LIN {X 0,Y 575.893,Z 1106.128,A -85,B 0,C 180,E1 20228.402,E2 20228.402} C_VEL
LIN {X 0,Y 578.191,Z 1090.768,A -85,B 0,C 180,E1 20226.346,E2 20226.346} C_VEL
LIN {X 0,Y 580.577,Z 1075.313,A -85,B 0,C 180,E1 20224.483,E2 20224.483} C_VEL
LIN {X 0,Y 583.778,Z 1055.461,A -85,B 0,C 180,E1 20222.344,E2 20222.344} C_VEL
LIN {X 0,Y 586.979,Z 1035.406,A -85,B 0,C 180,E1 20220.459,E2 20220.459} C_VEL
LIN {X 0,Y 589.808,Z 1017.804,A -85,B 0,C 180,E1 20218.978,E2 20218.978} C_VEL
LIN {X 0,Y 592.773,Z 999.025,A -85,B 0,C 180,E1 20217.561,E2 20217.561} C_VEL
LIN {X 0,Y 596.383,Z 975.656,A -85,B 0,C 180,E1 20216.004,E2 20216.004} C_VEL
LIN {X 0,Y 599.713,Z 951.946,A -85,B 0,C 180,E1 20214.652,E2 20214.652} C_VEL
LIN {X 0,Y 602.211,Z 933.032,A -85,B 0,C 180,E1 20213.707,E2 20213.707} C_VEL
LIN {X 0,Y 604.654,Z 912.644,A -85,B 0,C 180,E1 20212.814,E2 20212.814} C_VEL
LIN {X 0,Y 607.042,Z 890.934,A -85,B 0,C 180,E1 20212.003,E2 20212.003} C_VEL
LIN {X 0,Y 609.575,Z 864.282,A -85,B 0,C 180,E1 20211.183,E2 20211.183} C_VEL
LIN {X 0,Y 611.456,Z 838.408,A -85,B 0,C 180,E1 20210.573,E2 20210.573} C_VEL
LIN {X 0,Y 612.734,Z 815.587,A -85,B 0,C 180,E1 20210.167,E2 20210.167} C_VEL
LIN {X 0,Y 618.857,Z 603.625,A -85,B 0,C 180,E1 20207.181,E2 20207.181} C_VEL
LIN {X 0,Y 624.347,Z 417.468,A -85,B 0,C 180,E1 20204.512,E2 20204.512} C_VEL
LIN {X 0,Y 610.025,Z 396.851,A -85,B 0,C 180,E1 20202.474,E2 20202.474} C_VEL
LIN {X 0,Y 593.081,Z 373.946,A -85,B 0,C 180,E1 20199.872,E2 20199.872} C_VEL
LIN {X 0,Y 586.63,Z 365.779,A -85,B 0,C 180,E1 20198.816,E2 20198.816} C_VEL
LIN {X 0,Y 582.842,Z 360.939,A -85,B 0,C 180,E1 20198.172,E2 20198.172} C_VEL
LIN {X 0,Y 579.584,Z 357.07,A -85,B 0,C 180,E1 20197.61,E2 20197.61} C_VEL
LIN {X 0,Y 578.5,Z 355.414,A -85,B 0,C 180,E1 20197.412,E2 20197.412} C_VEL
LIN {X 0,Y 575.382,Z 352.205,A -85,B 0,C 180,E1 20196.868,E2 20196.868} C_VEL
LIN {X 0,Y 573.879,Z 349.556,A -85,B 0,C 180,E1 20196.576,E2 20196.576} C_VEL
LIN {X 0,Y 571.012,Z 347.283,A -85,B 0,C 180,E1 20196.072,E2 20196.072} C_VEL
LIN {X 0,Y 569.539,Z 344.267,A -85,B 0,C 180,E1 20195.766,E2 20195.766} C_VEL
LIN {X 0,Y 569.361,Z 343.303,A -85,B 0,C 180,E1 20195.707,E2 20195.707} C_VEL
LIN {X 0,Y 569.351,Z 343.308,A -85,B 0,C 180,E1 20192.358,E2 20192.358} C_VEL
LIN {X 0,Y 569.387,Z 343.308,A -85,B 0,C 180,E1 20189.107,E2 20189.107} C_VEL
LIN {X 0,Y 569.334,Z 343.259,A -85,B 0,C 180,E1 20185.82,E2 20185.82} C_VEL
LIN {X 0,Y 569.37,Z 343.294,A -85,B 0,C 180,E1 20182.51,E2 20182.51} C_VEL
LIN {X 0,Y 569.339,Z 343.26,A -85,B 0,C 180,E1 20179.386,E2 20179.386} C_VEL
LIN {X 0,Y 569.332,Z 343.299,A -85,B 0,C 180,E1 20176.006,E2 20176.006} C_VEL
LIN {X 0,Y 569.365,Z 343.249,A -85,B 0,C 180,E1 20172.887,E2 20172.887} C_VEL
LIN {X 0,Y 569.32,Z 343.309,A -85,B 0,C 180,E1 20169.707,E2 20169.707} C_VEL
LIN {X 0,Y 569.387,Z 343.308,A -85,B 0,C 180,E1 20166.554,E2 20166.554} C_VEL
LIN {X 0,Y 569.312,Z 343.314,A -85,B 0,C 180,E1 20163.323,E2 20163.323} C_VEL
LIN {X 0,Y 569.356,Z 343.31,A -85,B 0,C 180,E1 20160.101,E2 20160.101} C_VEL
LIN {X 0,Y 569.307,Z 343.31,A -85,B 0,C 180,E1 20157.08,E2 20157.08} C_VEL
LIN {X 0,Y 569.321,Z 343.308,A -85,B 0,C 180,E1 20153.745,E2 20153.745} C_VEL
LIN {X 0,Y 569.3,Z 343.302,A -85,B 0,C 180,E1 20150.905,E2 20150.905} C_VEL
LIN {X 0,Y 569.305,Z 343.271,A -85,B 0,C 180,E1 20147.557,E2 20147.557} C_VEL
LIN {X 0,Y 569.299,Z 343.289,A -85,B 0,C 180,E1 20144.628,E2 20144.628} C_VEL
LIN {X 0,Y 569.287,Z 343.271,A -85,B 0,C 180,E1 20141.251,E2 20141.251} C_VEL
LIN {X 0,Y 569.315,Z 343.302,A -85,B 0,C 180,E1 20138.248,E2 20138.248} C_VEL
LIN {X 0,Y 569.275,Z 343.263,A -85,B 0,C 180,E1 20135,E2 20135} C_VEL
LIN {X 0,Y 569.359,Z 343.305,A -85,B 0,C 180,E1 20131.809,E2 20131.809} C_VEL
LIN {X 0,Y 569.297,Z 343.395,A -85,B 0,C 180,E1 20130.946,E2 20130.946} C_VEL
LIN {X 0,Y 570.439,Z 346.544,A -85,B 0,C 180,E1 20130.376,E2 20130.376} C_VEL
LIN {X 0,Y 571.962,Z 348.62,A -85,B 0,C 180,E1 20129.886,E2 20129.886} C_VEL
LIN {X 0,Y 574.856,Z 352.888,A -85,B 0,C 180,E1 20129.302,E2 20129.302} C_VEL
LIN {X 0,Y 577.63,Z 356.406,A -85,B 0,C 180,E1 20128.801,E2 20128.801} C_VEL
LIN {X 0,Y 584.527,Z 365.235,A -85,B 0,C 180,E1 20127.599,E2 20127.599} C_VEL
LIN {X 0,Y 592.875,Z 376.369,A -85,B 0,C 180,E1 20126.211,E2 20126.211} C_VEL
LIN {X 0,Y 606.926,Z 395.613,A -85,B 0,C 180,E1 20124.033,E2 20124.033} C_VEL
LIN {X 0,Y 619.297,Z 413.266,A -85,B 0,C 180,E1 20122.242,E2 20122.242} C_VEL
LIN {X 0,Y 624.456,Z 421.081,A -85,B 0,C 180,E1 20121.519,E2 20121.519} C_VEL
LIN {X 0,Y 618.456,Z 624.273,A -85,B 0,C 180,E1 20118.616,E2 20118.616} C_VEL
LIN {X 0,Y 612.63,Z 826.368,A -85,B 0,C 180,E1 20115.769,E2 20115.769} C_VEL
LIN {X 0,Y 611.284,Z 850.031,A -85,B 0,C 180,E1 20115.341,E2 20115.341} C_VEL
LIN {X 0,Y 609.041,Z 878.855,A -85,B 0,C 180,E1 20114.633,E2 20114.633} C_VEL
LIN {X 0,Y 606.975,Z 900.549,A -85,B 0,C 180,E1 20113.955,E2 20113.955} C_VEL
LIN {X 0,Y 604.717,Z 921.391,A -85,B 0,C 180,E1 20113.181,E2 20113.181} C_VEL
LIN {X 0,Y 602.477,Z 940.397,A -85,B 0,C 180,E1 20112.361,E2 20112.361} C_VEL
LIN {X 0,Y 599.946,Z 959.808,A -85,B 0,C 180,E1 20111.411,E2 20111.411} C_VEL
LIN {X 0,Y 597.021,Z 980.896,A -85,B 0,C 180,E1 20110.234,E2 20110.234} C_VEL
LIN {X 0,Y 593.329,Z 1005.625,A -85,B 0,C 180,E1 20108.636,E2 20108.636} C_VEL
LIN {X 0,Y 590.183,Z 1025.543,A -85,B 0,C 180,E1 20107.155,E2 20107.155} C_VEL
LIN {X 0,Y 587.381,Z 1042.971,A -85,B 0,C 180,E1 20105.709,E2 20105.709} C_VEL
LIN {X 0,Y 584.603,Z 1060.16,A -85,B 0,C 180,E1 20104.124,E2 20104.124} C_VEL
LIN {X 0,Y 581.464,Z 1079.866,A -85,B 0,C 180,E1 20102.097,E2 20102.097} C_VEL
LIN {X 0,Y 578.617,Z 1097.979,A -85,B 0,C 180,E1 20099.961,E2 20099.961} C_VEL
LIN {X 0,Y 576.364,Z 1112.967,A -85,B 0,C 180,E1 20097.99,E2 20097.99} C_VEL
LIN {X 0,Y 574.255,Z 1127.876,A -85,B 0,C 180,E1 20095.804,E2 20095.804} C_VEL
LIN {X 0,Y 572.237,Z 1143.699,A -85,B 0,C 180,E1 20093.151,E2 20093.151} C_VEL
LIN {X 0,Y 570.921,Z 1155.261,A -85,B 0,C 180,E1 20090.933,E2 20090.933} C_VEL
LIN {X 0,Y 569.926,Z 1165.441,A -85,B 0,C 180,E1 20088.727,E2 20088.727} C_VEL
LIN {X 0,Y 569.029,Z 1176.307,A -85,B 0,C 180,E1 20086.014,E2 20086.014} C_VEL
LIN {X 0,Y 568.478,Z 1185.168,A -85,B 0,C 180,E1 20083.322,E2 20083.322} C_VEL
LIN {X 0,Y 568.16,Z 1191.596,A -85,B 0,C 180,E1 20080.957,E2 20080.957} C_VEL
LIN {X 0,Y 568.007,Z 1197.191,A -85,B 0,C 180,E1 20078.381,E2 20078.381} C_VEL
LIN {X 0,Y 567.93,Z 1201.538,A -85,B 0,C 180,E1 20075.557,E2 20075.557} C_VEL
LIN {X 0,Y 567.917,Z 1203.848,A -85,B 0,C 180,E1 20073.129,E2 20073.129} C_VEL
LIN {X 0,Y 567.906,Z 1204.804,A -85,B 0,C 180,E1 20070.908,E2 20070.908} C_VEL
LIN {X 0,Y 567.916,Z 1204.736,A -85,B 0,C 180,E1 20068.79,E2 20068.79} C_VEL
LIN {X 0,Y 567.912,Z 1203.507,A -85,B 0,C 180,E1 20066.366,E2 20066.366} C_VEL
LIN {X 0,Y 567.948,Z 1200.336,A -85,B 0,C 180,E1 20063.531,E2 20063.531} C_VEL
LIN {X 0,Y 568.029,Z 1196.127,A -85,B 0,C 180,E1 20061.089,E2 20061.089} C_VEL
LIN {X 0,Y 568.191,Z 1190.834,A -85,B 0,C 180,E1 20058.736,E2 20058.736} C_VEL
LIN {X 0,Y 568.577,Z 1183.471,A -85,B 0,C 180,E1 20056.106,E2 20056.106} C_VEL
LIN {X 0,Y 569.205,Z 1173.921,A -85,B 0,C 180,E1 20053.362,E2 20053.362} C_VEL
LIN {X 0,Y 570.007,Z 1164.53,A -85,B 0,C 180,E1 20051.064,E2 20051.064} C_VEL
LIN {X 0,Y 571.043,Z 1154.241,A -85,B 0,C 180,E1 20048.857,E2 20048.857} C_VEL
LIN {X 0,Y 572.616,Z 1140.8,A -85,B 0,C 180,E1 20046.321,E2 20046.321} C_VEL
LIN {X 0,Y 574.532,Z 1125.781,A -85,B 0,C 180,E1 20043.877,E2 20043.877} C_VEL
LIN {X 0,Y 576.537,Z 1111.839,A -85,B 0,C 180,E1 20041.854,E2 20041.854} C_VEL
LIN {X 0,Y 579.025,Z 1095.328,A -85,B 0,C 180,E1 20039.704,E2 20039.704} C_VEL
LIN {X 0,Y 582.168,Z 1075.368,A -85,B 0,C 180,E1 20037.428,E2 20037.428} C_VEL
LIN {X 0,Y 584.782,Z 1059.048,A -85,B 0,C 180,E1 20035.769,E2 20035.769} C_VEL
LIN {X 0,Y 587.478,Z 1042.379,A -85,B 0,C 180,E1 20034.24,E2 20034.24} C_VEL
LIN {X 0,Y 590.374,Z 1024.365,A -85,B 0,C 180,E1 20032.752,E2 20032.752} C_VEL
LIN {X 0,Y 594.05,Z 1001.024,A -85,B 0,C 180,E1 20031.044,E2 20031.044} C_VEL
LIN {X 0,Y 597.217,Z 979.4,A -85,B 0,C 180,E1 20029.678,E2 20029.678} C_VEL
LIN {X 0,Y 599.974,Z 959.58,A -85,B 0,C 180,E1 20028.578,E2 20028.578} C_VEL
LIN {X 0,Y 602.471,Z 940.399,A -85,B 0,C 180,E1 20027.639,E2 20027.639} C_VEL
LIN {X 0,Y 604.751,Z 921.029,A -85,B 0,C 180,E1 20026.805,E2 20026.805} C_VEL
LIN {X 0,Y 607.072,Z 899.565,A -85,B 0,C 180,E1 20026.012,E2 20026.012} C_VEL
LIN {X 0,Y 609.587,Z 872.897,A -85,B 0,C 180,E1 20025.2,E2 20025.2} C_VEL
LIN {X 0,Y 611.441,Z 847.173,A -85,B 0,C 180,E1 20024.602,E2 20024.602} C_VEL
LIN {X 0,Y 612.679,Z 825.072,A -85,B 0,C 180,E1 20024.212,E2 20024.212} C_VEL
LIN {X 0,Y 618.751,Z 613.717,A -85,B 0,C 180,E1 20021.235,E2 20021.235} C_VEL
LIN {X 0,Y 624.752,Z 420.897,A -85,B 0,C 180,E1 20018.456,E2 20018.456} C_VEL
LIN {X 0,Y 613.139,Z 403.007,A -85,B 0,C 180,E1 20016.646,E2 20016.646} C_VEL
LIN {X 0,Y 603.928,Z 389.594,A -85,B 0,C 180,E1 20015.094,E2 20015.094} C_VEL
LIN {X 0,Y 596.914,Z 380.267,A -85,B 0,C 180,E1 20013.847,E2 20013.847} C_VEL
LIN {X 0,Y 592.314,Z 374.199,A -85,B 0,C 180,E1 20012.985,E2 20012.985} C_VEL
LIN {X 0,Y 588.72,Z 369.537,A -85,B 0,C 180,E1 20012.287,E2 20012.287} C_VEL
LIN {X 0,Y 581.129,Z 359.893,A -85,B 0,C 180,E1 20010.732,E2 20010.732} C_VEL
LIN {X 0,Y 577.588,Z 355.415,A -85,B 0,C 180,E1 20009.963,E2 20009.963} C_VEL
LIN {X 0,Y 572.996,Z 350.191,A -85,B 0,C 180,E1 20008.935,E2 20008.935} C_VEL
LIN {X 0,Y 571.907,Z 348.267,A -85,B 0,C 180,E1 20008.623,E2 20008.623} C_VEL
LIN {X 0,Y 569.741,Z 345.073,A -85,B 0,C 180,E1 20007.715,E2 20007.715} C_VEL
LIN {X 0,Y 569.286,Z 343.283,A -85,B 0,C 180,E1 20007.288,E2 20007.288} C_VEL
LIN {X 0,Y 569.359,Z 343.309,A -85,B 0,C 180,E1 20004.154,E2 20004.154} C_VEL
LIN {X 0,Y 569.278,Z 343.275,A -85,B 0,C 180,E1 20001.104,E2 20001.104} C_VEL
LIN {X 0,Y 569.349,Z 343.283,A -85,B 0,C 180,E1 19998.005,E2 19998.005} C_VEL
LIN {X 0,Y 569.274,Z 343.303,A -85,B 0,C 180,E1 19994.859,E2 19994.859} C_VEL
LIN {X 0,Y 569.343,Z 343.264,A -85,B 0,C 180,E1 19991.755,E2 19991.755} C_VEL
LIN {X 0,Y 569.28,Z 343.319,A -85,B 0,C 180,E1 19988.688,E2 19988.688} C_VEL
LIN {X 0,Y 569.343,Z 343.262,A -85,B 0,C 180,E1 19985.543,E2 19985.543} C_VEL
LIN {X 0,Y 569.291,Z 343.312,A -85,B 0,C 180,E1 19982.416,E2 19982.416} C_VEL
LIN {X 0,Y 569.316,Z 343.278,A -85,B 0,C 180,E1 19979.094,E2 19979.094} C_VEL
LIN {X 0,Y 569.298,Z 343.287,A -85,B 0,C 180,E1 19976.173,E2 19976.173} C_VEL
LIN {X 0,Y 569.308,Z 343.307,A -85,B 0,C 180,E1 19972.735,E2 19972.735} C_VEL
LIN {X 0,Y 569.322,Z 343.267,A -85,B 0,C 180,E1 19969.782,E2 19969.782} C_VEL
LIN {X 0,Y 569.31,Z 343.313,A -85,B 0,C 180,E1 19966.491,E2 19966.491} C_VEL
LIN {X 0,Y 569.346,Z 343.269,A -85,B 0,C 180,E1 19963.471,E2 19963.471} C_VEL
LIN {X 0,Y 569.31,Z 343.275,A -85,B 0,C 180,E1 19960.282,E2 19960.282} C_VEL
LIN {X 0,Y 569.336,Z 343.46,A -85,B 0,C 180,E1 19957.795,E2 19957.795} C_VEL
LIN {X 0,Y 570.347,Z 346.325,A -85,B 0,C 180,E1 19957.504,E2 19957.504} C_VEL
LIN {X 0,Y 572.829,Z 348.93,A -85,B 0,C 180,E1 19956.929,E2 19956.929} C_VEL
LIN {X 0,Y 574.665,Z 350.184,A -85,B 0,C 180,E1 19956.532,E2 19956.532} C_VEL
LIN {X 0,Y 576.844,Z 353.797,A -85,B 0,C 180,E1 19956.016,E2 19956.016} C_VEL
LIN {X 0,Y 579.949,Z 356.442,A -85,B 0,C 180,E1 19955.367,E2 19955.367} C_VEL
LIN {X 0,Y 582.737,Z 360.467,A -85,B 0,C 180,E1 19954.761,E2 19954.761} C_VEL
LIN {X 0,Y 585.167,Z 362.766,A -85,B 0,C 180,E1 19954.277,E2 19954.277} C_VEL
LIN {X 0,Y 588.549,Z 367.081,A -85,B 0,C 180,E1 19953.596,E2 19953.596} C_VEL
LIN {X 0,Y 597.415,Z 378.223,A -85,B 0,C 180,E1 19951.918,E2 19951.918} C_VEL
LIN {X 0,Y 605.947,Z 389.787,A -85,B 0,C 180,E1 19950.409,E2 19950.409} C_VEL
LIN {X 0,Y 614.074,Z 401.365,A -85,B 0,C 180,E1 19949.06,E2 19949.06} C_VEL
LIN {X 0,Y 624.696,Z 417.64,A -85,B 0,C 180,E1 19947.41,E2 19947.41} C_VEL
LIN {X 0,Y 617.818,Z 639.221,A -85,B 0,C 180,E1 19944.226,E2 19944.226} C_VEL
LIN {X 0,Y 614.71,Z 749.255,A -85,B 0,C 180,E1 19942.68,E2 19942.68} C_VEL
LIN {X 0,Y 613.809,Z 756.956,A -85,B 0,C 180,E1 19942.64,E2 19942.64} C_VEL
LIN {X 0,Y 608.934,Z 777.584,A -85,B 0,C 180,E1 19942.779,E2 19942.779} C_VEL
LIN {X 0,Y 608.218,Z 784.192,A -85,B 0,C 180,E1 19942.739,E2 19942.739} C_VEL
LIN {X 0,Y 606.695,Z 825.935,A -85,B 0,C 180,E1 19942.121,E2 19942.121} C_VEL
LIN {X 0,Y 604.803,Z 852.528,A -85,B 0,C 180,E1 19941.563,E2 19941.563} C_VEL
LIN {X 0,Y 602.859,Z 874.596,A -85,B 0,C 180,E1 19940.97,E2 19940.97} C_VEL
LIN {X 0,Y 600.68,Z 896.035,A -85,B 0,C 180,E1 19940.266,E2 19940.266} C_VEL
LIN {X 0,Y 597.724,Z 921.458,A -85,B 0,C 180,E1 19939.268,E2 19939.268} C_VEL
LIN {X 0,Y 594.254,Z 947.046,A -85,B 0,C 180,E1 19938.047,E2 19938.047} C_VEL
LIN {X 0,Y 591.224,Z 967.695,A -85,B 0,C 180,E1 19936.901,E2 19936.901} C_VEL
LIN {X 0,Y 588.099,Z 987.768,A -85,B 0,C 180,E1 19935.637,E2 19935.637} C_VEL
LIN {X 0,Y 584.168,Z 1012.057,A -85,B 0,C 180,E1 19933.884,E2 19933.884} C_VEL
LIN {X 0,Y 580.824,Z 1031.805,A -85,B 0,C 180,E1 19932.247,E2 19932.247} C_VEL
LIN {X 0,Y 577.972,Z 1048.487,A -85,B 0,C 180,E1 19930.707,E2 19930.707} C_VEL
LIN {X 0,Y 575.229,Z 1064.617,A -85,B 0,C 180,E1 19929.057,E2 19929.057} C_VEL
LIN {X 0,Y 572.159,Z 1083.109,A -85,B 0,C 180,E1 19926.952,E2 19926.952} C_VEL
LIN {X 0,Y 569.347,Z 1100.558,A -85,B 0,C 180,E1 19924.68,E2 19924.68} C_VEL
LIN {X 0,Y 567.145,Z 1114.998,A -85,B 0,C 180,E1 19922.57,E2 19922.57} C_VEL
LIN {X 0,Y 565.18,Z 1129.015,A -85,B 0,C 180,E1 19920.278,E2 19920.278} C_VEL
LIN {X 0,Y 563.324,Z 1143.865,A -85,B 0,C 180,E1 19917.483,E2 19917.483} C_VEL
LIN {X 0,Y 562.209,Z 1154.097,A -85,B 0,C 180,E1 19915.266,E2 19915.266} C_VEL
LIN {X 0,Y 561.345,Z 1163.439,A -85,B 0,C 180,E1 19912.959,E2 19912.959} C_VEL
LIN {X 0,Y 560.664,Z 1172.891,A -85,B 0,C 180,E1 19910.241,E2 19910.241} C_VEL
LIN {X 0,Y 560.237,Z 1180.671,A -85,B 0,C 180,E1 19907.447,E2 19907.447} C_VEL
LIN {X 0,Y 560.043,Z 1185.895,A -85,B 0,C 180,E1 19905.109,E2 19905.109} C_VEL
LIN {X 0,Y 559.95,Z 1190.068,A -85,B 0,C 180,E1 19902.687,E2 19902.687} C_VEL
LIN {X 0,Y 559.914,Z 1193.254,A -85,B 0,C 180,E1 19899.975,E2 19899.975} C_VEL
LIN {X 0,Y 559.914,Z 1194.691,A -85,B 0,C 180,E1 19897.387,E2 19897.387} C_VEL
LIN {X 0,Y 559.904,Z 1194.824,A -85,B 0,C 180,E1 19895.122,E2 19895.122} C_VEL
LIN {X 0,Y 559.911,Z 1193.901,A -85,B 0,C 180,E1 19892.866,E2 19892.866} C_VEL
LIN {X 0,Y 559.929,Z 1191.749,A -85,B 0,C 180,E1 19890.511,E2 19890.511} C_VEL
LIN {X 0,Y 560.001,Z 1187.917,A -85,B 0,C 180,E1 19887.851,E2 19887.851} C_VEL
LIN {X 0,Y 560.158,Z 1182.188,A -85,B 0,C 180,E1 19885.085,E2 19885.085} C_VEL
LIN {X 0,Y 560.481,Z 1175.927,A -85,B 0,C 180,E1 19882.704,E2 19882.704} C_VEL
LIN {X 0,Y 560.966,Z 1168.152,A -85,B 0,C 180,E1 19880.251,E2 19880.251} C_VEL
LIN {X 0,Y 561.886,Z 1157.613,A -85,B 0,C 180,E1 19877.461,E2 19877.461} C_VEL
LIN {X 0,Y 563.013,Z 1146.479,A -85,B 0,C 180,E1 19874.972,E2 19874.972} C_VEL
LIN {X 0,Y 564.367,Z 1135.127,A -85,B 0,C 180,E1 19872.737,E2 19872.737} C_VEL
LIN {X 0,Y 566.369,Z 1120.464,A -85,B 0,C 180,E1 19870.186,E2 19870.186} C_VEL
LIN {X 0,Y 568.722,Z 1104.546,A -85,B 0,C 180,E1 19867.79,E2 19867.79} C_VEL
LIN {X 0,Y 571.033,Z 1089.852,A -85,B 0,C 180,E1 19865.812,E2 19865.812} C_VEL
LIN {X 0,Y 573.876,Z 1072.651,A -85,B 0,C 180,E1 19863.733,E2 19863.733} C_VEL
LIN {X 0,Y 577.452,Z 1051.608,A -85,B 0,C 180,E1 19861.508,E2 19861.508} C_VEL
LIN {X 0,Y 580.343,Z 1034.596,A -85,B 0,C 180,E1 19859.909,E2 19859.909} C_VEL
LIN {X 0,Y 583.214,Z 1017.629,A -85,B 0,C 180,E1 19858.473,E2 19858.473} C_VEL
LIN {X 0,Y 586.21,Z 999.533,A -85,B 0,C 180,E1 19857.094,E2 19857.094} C_VEL
LIN {X 0,Y 589.867,Z 977.086,A -85,B 0,C 180,E1 19855.576,E2 19855.576} C_VEL
LIN {X 0,Y 593.49,Z 952.586,A -85,B 0,C 180,E1 19854.159,E2 19854.159} C_VEL
LIN {X 0,Y 596.234,Z 932.77,A -85,B 0,C 180,E1 19853.164,E2 19853.164} C_VEL
LIN {X 0,Y 598.786,Z 912.329,A -85,B 0,C 180,E1 19852.266,E2 19852.266} C_VEL
LIN {X 0,Y 601.358,Z 889.817,A -85,B 0,C 180,E1 19851.427,E2 19851.427} C_VEL
LIN {X 0,Y 604.064,Z 861.722,A -85,B 0,C 180,E1 19850.576,E2 19850.576} C_VEL
LIN {X 0,Y 605.893,Z 837.476,A -85,B 0,C 180,E1 19850.012,E2 19850.012} C_VEL
LIN {X 0,Y 607.192,Z 814.887,A -85,B 0,C 180,E1 19849.614,E2 19849.614} C_VEL
LIN {X 0,Y 613.675,Z 600.595,A -85,B 0,C 180,E1 19846.574,E2 19846.574} C_VEL
LIN {X 0,Y 619.157,Z 421.501,A -85,B 0,C 180,E1 19843.998,E2 19843.998} C_VEL
LIN {X 0,Y 605.718,Z 402.239,A -85,B 0,C 180,E1 19842.051,E2 19842.051} C_VEL
LIN {X 0,Y 589.573,Z 380.211,A -85,B 0,C 180,E1 19839.525,E2 19839.525} C_VEL
LIN {X 0,Y 583.559,Z 372.546,A -85,B 0,C 180,E1 19838.524,E2 19838.524} C_VEL
LIN {X 0,Y 579.54,Z 367.518,A -85,B 0,C 180,E1 19837.832,E2 19837.832} C_VEL
LIN {X 0,Y 575.973,Z 362.901,A -85,B 0,C 180,E1 19837.198,E2 19837.198} C_VEL
LIN {X 0,Y 572.053,Z 358.443,A -85,B 0,C 180,E1 19836.493,E2 19836.493} C_VEL
LIN {X 0,Y 570.76,Z 356.543,A -85,B 0,C 180,E1 19836.246,E2 19836.246} C_VEL
LIN {X 0,Y 567.726,Z 353.563,A -85,B 0,C 180,E1 19835.691,E2 19835.691} C_VEL
LIN {X 0,Y 566.052,Z 350.576,A -85,B 0,C 180,E1 19835.346,E2 19835.346} C_VEL
LIN {X 0,Y 563.155,Z 348.335,A -85,B 0,C 180,E1 19834.808,E2 19834.808} C_VEL
LIN {X 0,Y 561.648,Z 345.45,A -85,B 0,C 180,E1 19834.481,E2 19834.481} C_VEL
LIN {X 0,Y 561.415,Z 344.305,A -85,B 0,C 180,E1 19834.404,E2 19834.404} C_VEL
LIN {X 0,Y 561.444,Z 344.287,A -85,B 0,C 180,E1 19831.096,E2 19831.096} C_VEL
LIN {X 0,Y 561.397,Z 344.265,A -85,B 0,C 180,E1 19827.932,E2 19827.932} C_VEL
LIN {X 0,Y 561.434,Z 344.27,A -85,B 0,C 180,E1 19824.629,E2 19824.629} C_VEL
LIN {X 0,Y 561.396,Z 344.253,A -85,B 0,C 180,E1 19821.525,E2 19821.525} C_VEL
LIN {X 0,Y 561.396,Z 344.285,A -85,B 0,C 180,E1 19818.054,E2 19818.054} C_VEL
LIN {X 0,Y 561.437,Z 344.24,A -85,B 0,C 180,E1 19814.86,E2 19814.86} C_VEL
LIN {X 0,Y 561.38,Z 344.279,A -85,B 0,C 180,E1 19811.59,E2 19811.59} C_VEL
LIN {X 0,Y 561.437,Z 344.282,A -85,B 0,C 180,E1 19808.397,E2 19808.397} C_VEL
LIN {X 0,Y 561.374,Z 344.287,A -85,B 0,C 180,E1 19805.314,E2 19805.314} C_VEL
LIN {X 0,Y 561.405,Z 344.286,A -85,B 0,C 180,E1 19802.041,E2 19802.041} C_VEL
LIN {X 0,Y 561.373,Z 344.301,A -85,B 0,C 180,E1 19799.081,E2 19799.081} C_VEL
LIN {X 0,Y 561.38,Z 344.297,A -85,B 0,C 180,E1 19795.71,E2 19795.71} C_VEL
LIN {X 0,Y 561.379,Z 344.304,A -85,B 0,C 180,E1 19792.735,E2 19792.735} C_VEL
LIN {X 0,Y 561.363,Z 344.304,A -85,B 0,C 180,E1 19789.428,E2 19789.428} C_VEL
LIN {X 0,Y 561.396,Z 344.238,A -85,B 0,C 180,E1 19786.297,E2 19786.297} C_VEL
LIN {X 0,Y 561.348,Z 344.307,A -85,B 0,C 180,E1 19783.122,E2 19783.122} C_VEL
LIN {X 0,Y 561.407,Z 344.241,A -85,B 0,C 180,E1 19780.004,E2 19780.004} C_VEL
LIN {X 0,Y 561.339,Z 344.299,A -85,B 0,C 180,E1 19776.929,E2 19776.929} C_VEL
LIN {X 0,Y 561.407,Z 344.251,A -85,B 0,C 180,E1 19773.788,E2 19773.788} C_VEL
LIN {X 0,Y 561.4,Z 344.469,A -85,B 0,C 180,E1 19772.137,E2 19772.137} C_VEL
LIN {X 0,Y 562.81,Z 347.945,A -85,B 0,C 180,E1 19771.451,E2 19771.451} C_VEL
LIN {X 0,Y 564.29,Z 349.804,A -85,B 0,C 180,E1 19771.07,E2 19771.07} C_VEL
LIN {X 0,Y 567.253,Z 353.881,A -85,B 0,C 180,E1 19770.484,E2 19770.484} C_VEL
LIN {X 0,Y 569.152,Z 355.931,A -85,B 0,C 180,E1 19770.128,E2 19770.128} C_VEL
LIN {X 0,Y 572.695,Z 360.494,A -85,B 0,C 180,E1 19769.465,E2 19769.465} C_VEL
LIN {X 0,Y 585.667,Z 377.578,A -85,B 0,C 180,E1 19767.176,E2 19767.176} C_VEL
LIN {X 0,Y 599.164,Z 396.072,A -85,B 0,C 180,E1 19764.994,E2 19764.994} C_VEL
LIN {X 0,Y 615.014,Z 418.598,A -85,B 0,C 180,E1 19762.639,E2 19762.639} C_VEL
LIN {X 0,Y 619.242,Z 425.189,A -85,B 0,C 180,E1 19762.033,E2 19762.033} C_VEL
LIN {X 0,Y 612.98,Z 630.051,A -85,B 0,C 180,E1 19759.095,E2 19759.095} C_VEL
LIN {X 0,Y 607.041,Z 826.349,A -85,B 0,C 180,E1 19756.311,E2 19756.311} C_VEL
LIN {X 0,Y 605.628,Z 850.135,A -85,B 0,C 180,E1 19755.879,E2 19755.879} C_VEL
LIN {X 0,Y 603.298,Z 878.838,A -85,B 0,C 180,E1 19755.169,E2 19755.169} C_VEL
LIN {X 0,Y 601.066,Z 901.176,A -85,B 0,C 180,E1 19754.467,E2 19754.467} C_VEL
LIN {X 0,Y 598.69,Z 922.091,A -85,B 0,C 180,E1 19753.683,E2 19753.683} C_VEL
LIN {X 0,Y 596.295,Z 941.417,A -85,B 0,C 180,E1 19752.84,E2 19752.84} C_VEL
LIN {X 0,Y 593.55,Z 961.475,A -85,B 0,C 180,E1 19751.843,E2 19751.843} C_VEL
LIN {X 0,Y 589.933,Z 986.302,A -85,B 0,C 180,E1 19750.42,E2 19750.42} C_VEL
LIN {X 0,Y 586.379,Z 1008.478,A -85,B 0,C 180,E1 19748.935,E2 19748.935} C_VEL
LIN {X 0,Y 583.453,Z 1026.209,A -85,B 0,C 180,E1 19747.596,E2 19747.596} C_VEL
LIN {X 0,Y 580.566,Z 1043.294,A -85,B 0,C 180,E1 19746.161,E2 19746.161} C_VEL
LIN {X 0,Y 577.693,Z 1060.149,A -85,B 0,C 180,E1 19744.591,E2 19744.591} C_VEL
LIN {X 0,Y 574.375,Z 1079.866,A -85,B 0,C 180,E1 19742.542,E2 19742.542} C_VEL
LIN {X 0,Y 571.314,Z 1098.124,A -85,B 0,C 180,E1 19740.364,E2 19740.364} C_VEL
LIN {X 0,Y 569.023,Z 1112.601,A -85,B 0,C 180,E1 19738.438,E2 19738.438} C_VEL
LIN {X 0,Y 566.889,Z 1126.664,A -85,B 0,C 180,E1 19736.359,E2 19736.359} C_VEL
LIN {X 0,Y 564.72,Z 1142.542,A -85,B 0,C 180,E1 19733.699,E2 19733.699} C_VEL
LIN {X 0,Y 563.225,Z 1154.745,A -85,B 0,C 180,E1 19731.342,E2 19731.342} C_VEL
LIN {X 0,Y 562.124,Z 1164.981,A -85,B 0,C 180,E1 19729.105,E2 19729.105} C_VEL
LIN {X 0,Y 561.222,Z 1175.133,A -85,B 0,C 180,E1 19726.563,E2 19726.563} C_VEL
LIN {X 0,Y 560.562,Z 1184.559,A -85,B 0,C 180,E1 19723.724,E2 19723.724} C_VEL
LIN {X 0,Y 560.206,Z 1191.084,A -85,B 0,C 180,E1 19721.323,E2 19721.323} C_VEL
LIN {X 0,Y 560.033,Z 1196.329,A -85,B 0,C 180,E1 19718.936,E2 19718.936} C_VEL
LIN {X 0,Y 559.945,Z 1200.782,A -85,B 0,C 180,E1 19716.254,E2 19716.254} C_VEL
LIN {X 0,Y 559.914,Z 1203.641,A -85,B 0,C 180,E1 19713.481,E2 19713.481} C_VEL
LIN {X 0,Y 559.916,Z 1204.736,A -85,B 0,C 180,E1 19711.228,E2 19711.228} C_VEL
LIN {X 0,Y 559.906,Z 1204.804,A -85,B 0,C 180,E1 19709.079,E2 19709.079} C_VEL
LIN {X 0,Y 559.916,Z 1203.845,A -85,B 0,C 180,E1 19706.827,E2 19706.827} C_VEL
LIN {X 0,Y 559.934,Z 1201.535,A -85,B 0,C 180,E1 19704.364,E2 19704.364} C_VEL
LIN {X 0,Y 560.017,Z 1197.151,A -85,B 0,C 180,E1 19701.478,E2 19701.478} C_VEL
LIN {X 0,Y 560.181,Z 1191.595,A -85,B 0,C 180,E1 19698.886,E2 19698.886} C_VEL
LIN {X 0,Y 560.531,Z 1185.078,A -85,B 0,C 180,E1 19696.456,E2 19696.456} C_VEL
LIN {X 0,Y 561.163,Z 1175.942,A -85,B 0,C 180,E1 19693.649,E2 19693.649} C_VEL
LIN {X 0,Y 562.082,Z 1165.446,A -85,B 0,C 180,E1 19691.003,E2 19691.003} C_VEL
LIN {X 0,Y 563.161,Z 1155.269,A -85,B 0,C 180,E1 19688.765,E2 19688.765} C_VEL
LIN {X 0,Y 564.639,Z 1143.132,A -85,B 0,C 180,E1 19686.409,E2 19686.409} C_VEL
LIN {X 0,Y 566.813,Z 1127.18,A -85,B 0,C 180,E1 19683.72,E2 19683.72} C_VEL
LIN {X 0,Y 569.021,Z 1112.607,A -85,B 0,C 180,E1 19681.563,E2 19681.563} C_VEL
LIN {X 0,Y 571.337,Z 1097.983,A -85,B 0,C 180,E1 19679.618,E2 19679.618} C_VEL
LIN {X 0,Y 574.601,Z 1078.506,A -85,B 0,C 180,E1 19677.312,E2 19677.312} C_VEL
LIN {X 0,Y 577.785,Z 1059.602,A -85,B 0,C 180,E1 19675.356,E2 19675.356} C_VEL
LIN {X 0,Y 580.645,Z 1042.82,A -85,B 0,C 180,E1 19673.798,E2 19673.798} C_VEL
LIN {X 0,Y 583.45,Z 1026.21,A -85,B 0,C 180,E1 19672.405,E2 19672.405} C_VEL
LIN {X 0,Y 586.487,Z 1007.814,A -85,B 0,C 180,E1 19671.017,E2 19671.017} C_VEL
LIN {X 0,Y 590.303,Z 983.798,A -85,B 0,C 180,E1 19669.426,E2 19669.426} C_VEL
LIN {X 0,Y 593.657,Z 960.626,A -85,B 0,C 180,E1 19668.113,E2 19668.113} C_VEL
LIN {X 0,Y 596.289,Z 941.407,A -85,B 0,C 180,E1 19667.161,E2 19667.161} C_VEL
LIN {X 0,Y 598.68,Z 922.085,A -85,B 0,C 180,E1 19666.318,E2 19666.318} C_VEL
LIN {X 0,Y 601.058,Z 901.159,A -85,B 0,C 180,E1 19665.534,E2 19665.534} C_VEL
LIN {X 0,Y 603.301,Z 878.702,A -85,B 0,C 180,E1 19664.828,E2 19664.828} C_VEL
LIN {X 0,Y 605.639,Z 849.775,A -85,B 0,C 180,E1 19664.115,E2 19664.115} C_VEL
LIN {X 0,Y 607.038,Z 826.18,A -85,B 0,C 180,E1 19663.688,E2 19663.688} C_VEL
LIN {X 0,Y 613.563,Z 612.315,A -85,B 0,C 180,E1 19660.647,E2 19660.647} C_VEL
LIN {X 0,Y 619.755,Z 424.952,A -85,B 0,C 180,E1 19657.923,E2 19657.923} C_VEL
LIN {X 0,Y 609.043,Z 408.278,A -85,B 0,C 180,E1 19656.201,E2 19656.201} C_VEL
LIN {X 0,Y 600.201,Z 395.388,A -85,B 0,C 180,E1 19654.675,E2 19654.675} C_VEL
LIN {X 0,Y 593.754,Z 386.715,A -85,B 0,C 180,E1 19653.5,E2 19653.5} C_VEL
LIN {X 0,Y 586.666,Z 377.187,A -85,B 0,C 180,E1 19652.125,E2 19652.125} C_VEL
LIN {X 0,Y 578.061,Z 366.414,A -85,B 0,C 180,E1 19650.337,E2 19650.337} C_VEL
LIN {X 0,Y 573.952,Z 361.201,A -85,B 0,C 180,E1 19649.421,E2 19649.421} C_VEL
LIN {X 0,Y 570.464,Z 357.088,A -85,B 0,C 180,E1 19648.617,E2 19648.617} C_VEL
LIN {X 0,Y 569.219,Z 355.332,A -85,B 0,C 180,E1 19648.313,E2 19648.313} C_VEL
LIN {X 0,Y 565.554,Z 351.283,A -85,B 0,C 180,E1 19647.423,E2 19647.423} C_VEL
LIN {X 0,Y 564.272,Z 349.512,A -85,B 0,C 180,E1 19647.091,E2 19647.091} C_VEL
LIN {X 0,Y 562.677,Z 347.738,A -85,B 0,C 180,E1 19646.603,E2 19646.603} C_VEL
LIN {X 0,Y 561.369,Z 344.261,A -85,B 0,C 180,E1 19645.704,E2 19645.704} C_VEL
LIN {X 0,Y 561.354,Z 344.272,A -85,B 0,C 180,E1 19642.738,E2 19642.738} C_VEL
LIN {X 0,Y 561.352,Z 344.307,A -85,B 0,C 180,E1 19639.348,E2 19639.348} C_VEL
LIN {X 0,Y 561.375,Z 344.254,A -85,B 0,C 180,E1 19636.258,E2 19636.258} C_VEL
LIN {X 0,Y 561.341,Z 344.29,A -85,B 0,C 180,E1 19633.075,E2 19633.075} C_VEL
LIN {X 0,Y 561.399,Z 344.268,A -85,B 0,C 180,E1 19629.949,E2 19629.949} C_VEL
LIN {X 0,Y 561.343,Z 344.267,A -85,B 0,C 180,E1 19626.854,E2 19626.854} C_VEL
LIN {X 0,Y 561.417,Z 344.29,A -85,B 0,C 180,E1 19623.676,E2 19623.676} C_VEL
LIN {X 0,Y 561.347,Z 344.255,A -85,B 0,C 180,E1 19620.51,E2 19620.51} C_VEL
LIN {X 0,Y 561.411,Z 344.299,A -85,B 0,C 180,E1 19617.32,E2 19617.32} C_VEL
LIN {X 0,Y 561.356,Z 344.257,A -85,B 0,C 180,E1 19614.173,E2 19614.173} C_VEL
LIN {X 0,Y 561.383,Z 344.275,A -85,B 0,C 180,E1 19610.879,E2 19610.879} C_VEL
LIN {X 0,Y 561.385,Z 344.281,A -85,B 0,C 180,E1 19607.763,E2 19607.763} C_VEL
LIN {X 0,Y 561.37,Z 344.253,A -85,B 0,C 180,E1 19604.49,E2 19604.49} C_VEL
LIN {X 0,Y 561.421,Z 344.282,A -85,B 0,C 180,E1 19601.346,E2 19601.346} C_VEL
LIN {X 0,Y 561.418,Z 344.404,A -85,B 0,C 180,E1 19599.501,E2 19599.501} C_VEL
LIN {X 0,Y 562.38,Z 347.155,A -85,B 0,C 180,E1 19599.197,E2 19599.197} C_VEL
LIN {X 0,Y 564.874,Z 349.923,A -85,B 0,C 180,E1 19598.56,E2 19598.56} C_VEL
LIN {X 0,Y 566.86,Z 351.183,A -85,B 0,C 180,E1 19598.095,E2 19598.095} C_VEL
LIN {X 0,Y 568.951,Z 354.735,A -85,B 0,C 180,E1 19597.555,E2 19597.555} C_VEL
LIN {X 0,Y 572.291,Z 357.65,A -85,B 0,C 180,E1 19596.797,E2 19596.797} C_VEL
LIN {X 0,Y 575.042,Z 361.575,A -85,B 0,C 180,E1 19596.154,E2 19596.154} C_VEL
LIN {X 0,Y 577.578,Z 363.895,A -85,B 0,C 180,E1 19595.614,E2 19595.614} C_VEL
LIN {X 0,Y 580.795,Z 368.127,A -85,B 0,C 180,E1 19594.916,E2 19594.916} C_VEL
LIN {X 0,Y 582.858,Z 370.308,A -85,B 0,C 180,E1 19594.495,E2 19594.495} C_VEL
LIN {X 0,Y 588.543,Z 377.445,A -85,B 0,C 180,E1 19593.351,E2 19593.351} C_VEL
LIN {X 0,Y 594.78,Z 385.418,A -85,B 0,C 180,E1 19592.165,E2 19592.165} C_VEL
LIN {X 0,Y 602.879,Z 396.476,A -85,B 0,C 180,E1 19590.708,E2 19590.708} C_VEL
LIN {X 0,Y 610.791,Z 407.902,A -85,B 0,C 180,E1 19589.367,E2 19589.367} C_VEL
LIN {X 0,Y 619.718,Z 421.875,A -85,B 0,C 180,E1 19587.938,E2 19587.938} C_VEL
LIN {X 0,Y 612.392,Z 643.582,A -85,B 0,C 180,E1 19584.727,E2 19584.727} C_VEL
LIN {X 0,Y 608.218,Z 784.192,A -85,B 0,C 180,E1 19582.739,E2 19582.739} C_VEL
LIN {X 0,Y 607.302,Z 791.893,A -85,B 0,C 180,E1 19582.702,E2 19582.702} C_VEL
LIN {X 0,Y 602.302,Z 812.494,A -85,B 0,C 180,E1 19582.835,E2 19582.835} C_VEL
LIN {X 0,Y 601.479,Z 819.085,A -85,B 0,C 180,E1 19582.783,E2 19582.783} C_VEL
LIN {X 0,Y 599.71,Z 846.681,A -85,B 0,C 180,E1 19582.257,E2 19582.257} C_VEL
LIN {X 0,Y 597.417,Z 872.214,A -85,B 0,C 180,E1 19581.59,E2 19581.59} C_VEL
LIN {X 0,Y 595.201,Z 893.433,A -85,B 0,C 180,E1 19580.905,E2 19580.905} C_VEL
LIN {X 0,Y 592.678,Z 914.485,A -85,B 0,C 180,E1 19580.101,E2 19580.101} C_VEL
LIN {X 0,Y 589.637,Z 937.531,A -85,B 0,C 180,E1 19579.064,E2 19579.064} C_VEL
LIN {X 0,Y 585.683,Z 963.791,A -85,B 0,C 180,E1 19577.664,E2 19577.664} C_VEL
LIN {X 0,Y 582.442,Z 983.826,A -85,B 0,C 180,E1 19576.422,E2 19576.422} C_VEL
LIN {X 0,Y 579.192,Z 1002.962,A -85,B 0,C 180,E1 19575.083,E2 19575.083} C_VEL
LIN {X 0,Y 575.588,Z 1023.512,A -85,B 0,C 180,E1 19573.464,E2 19573.464} C_VEL
LIN {X 0,Y 571.602,Z 1045.716,A -85,B 0,C 180,E1 19571.459,E2 19571.459} C_VEL
LIN {X 0,Y 568.58,Z 1062.568,A -85,B 0,C 180,E1 19569.741,E2 19569.741} C_VEL
LIN {X 0,Y 565.788,Z 1078.374,A -85,B 0,C 180,E1 19567.951,E2 19567.951} C_VEL
LIN {X 0,Y 562.747,Z 1096.156,A -85,B 0,C 180,E1 19565.708,E2 19565.708} C_VEL
LIN {X 0,Y 559.946,Z 1113.156,A -85,B 0,C 180,E1 19563.243,E2 19563.243} C_VEL
LIN {X 0,Y 557.921,Z 1126.451,A -85,B 0,C 180,E1 19561.073,E2 19561.073} C_VEL
LIN {X 0,Y 556.132,Z 1139.557,A -85,B 0,C 180,E1 19558.67,E2 19558.67} C_VEL
LIN {X 0,Y 554.545,Z 1152.736,A -85,B 0,C 180,E1 19555.87,E2 19555.87} C_VEL
LIN {X 0,Y 553.558,Z 1162.244,A -85,B 0,C 180,E1 19553.527,E2 19553.527} C_VEL
LIN {X 0,Y 552.927,Z 1170.05,A -85,B 0,C 180,E1 19551.313,E2 19551.313} C_VEL
LIN {X 0,Y 552.416,Z 1177.652,A -85,B 0,C 180,E1 19548.794,E2 19548.794} C_VEL
LIN {X 0,Y 552.104,Z 1184.661,A -85,B 0,C 180,E1 19545.87,E2 19545.87} C_VEL
LIN {X 0,Y 551.976,Z 1189.125,A -85,B 0,C 180,E1 19543.402,E2 19543.402} C_VEL
LIN {X 0,Y 551.926,Z 1192.188,A -85,B 0,C 180,E1 19541.071,E2 19541.071} C_VEL
LIN {X 0,Y 551.914,Z 1194.187,A -85,B 0,C 180,E1 19538.648,E2 19538.648} C_VEL
LIN {X 0,Y 551.9,Z 1194.978,A -85,B 0,C 180,E1 19535.823,E2 19535.823} C_VEL
LIN {X 0,Y 551.911,Z 1194.091,A -85,B 0,C 180,E1 19533.115,E2 19533.115} C_VEL
LIN {X 0,Y 551.927,Z 1192.066,A -85,B 0,C 180,E1 19530.726,E2 19530.726} C_VEL
LIN {X 0,Y 551.974,Z 1188.868,A -85,B 0,C 180,E1 19528.339,E2 19528.339} C_VEL
LIN {X 0,Y 552.132,Z 1183.841,A -85,B 0,C 180,E1 19525.638,E2 19525.638} C_VEL
LIN {X 0,Y 552.474,Z 1176.826,A -85,B 0,C 180,E1 19522.826,E2 19522.826} C_VEL
LIN {X 0,Y 552.948,Z 1169.481,A -85,B 0,C 180,E1 19520.423,E2 19520.423} C_VEL
LIN {X 0,Y 553.673,Z 1161.247,A -85,B 0,C 180,E1 19518.119,E2 19518.119} C_VEL
LIN {X 0,Y 554.869,Z 1149.905,A -85,B 0,C 180,E1 19515.387,E2 19515.387} C_VEL
LIN {X 0,Y 556.442,Z 1136.991,A -85,B 0,C 180,E1 19512.753,E2 19512.753} C_VEL
LIN {X 0,Y 558.19,Z 1124.707,A -85,B 0,C 180,E1 19510.538,E2 19510.538} C_VEL
LIN {X 0,Y 560.633,Z 1108.888,A -85,B 0,C 180,E1 19508.004,E2 19508.004} C_VEL
LIN {X 0,Y 563.39,Z 1092.18,A -85,B 0,C 180,E1 19505.685,E2 19505.685} C_VEL
LIN {X 0,Y 566.01,Z 1076.971,A -85,B 0,C 180,E1 19503.792,E2 19503.792} C_VEL
LIN {X 0,Y 569.025,Z 1060.066,A -85,B 0,C 180,E1 19501.899,E2 19501.899} C_VEL
LIN {X 0,Y 573.105,Z 1037.45,A -85,B 0,C 180,E1 19499.674,E2 19499.674} C_VEL
LIN {X 0,Y 576.439,Z 1018.746,A -85,B 0,C 180,E1 19498.059,E2 19498.059} C_VEL
LIN {X 0,Y 579.45,Z 1001.502,A -85,B 0,C 180,E1 19496.72,E2 19496.72} C_VEL
LIN {X 0,Y 582.701,Z 982.336,A -85,B 0,C 180,E1 19495.391,E2 19495.391} C_VEL
LIN {X 0,Y 586.639,Z 958.066,A -85,B 0,C 180,E1 19493.916,E2 19493.916} C_VEL
LIN {X 0,Y 590.02,Z 934.643,A -85,B 0,C 180,E1 19492.711,E2 19492.711} C_VEL
LIN {X 0,Y 592.74,Z 913.885,A -85,B 0,C 180,E1 19491.784,E2 19491.784} C_VEL
LIN {X 0,Y 595.257,Z 892.925,A -85,B 0,C 180,E1 19490.988,E2 19490.988} C_VEL
LIN {X 0,Y 597.587,Z 870.632,A -85,B 0,C 180,E1 19490.275,E2 19490.275} C_VEL
LIN {X 0,Y 599.999,Z 842.644,A -85,B 0,C 180,E1 19489.566,E2 19489.566} C_VEL
LIN {X 0,Y 601.54,Z 817.753,A -85,B 0,C 180,E1 19489.105,E2 19489.105} C_VEL
LIN {X 0,Y 606.201,Z 671.611,A -85,B 0,C 180,E1 19487.017,E2 19487.017} C_VEL
LIN {X 0,Y 613.146,Z 453.019,A -85,B 0,C 180,E1 19483.881,E2 19483.881} C_VEL
LIN {X 0,Y 613.941,Z 425.486,A -85,B 0,C 180,E1 19483.469,E2 19483.469} C_VEL
LIN {X 0,Y 601.013,Z 407.04,A -85,B 0,C 180,E1 19481.559,E2 19481.559} C_VEL
LIN {X 0,Y 586.082,Z 386.47,A -85,B 0,C 180,E1 19479.174,E2 19479.174} C_VEL
LIN {X 0,Y 580.119,Z 378.873,A -85,B 0,C 180,E1 19478.164,E2 19478.164} C_VEL
LIN {X 0,Y 576.261,Z 374.051,A -85,B 0,C 180,E1 19477.489,E2 19477.489} C_VEL
LIN {X 0,Y 571.86,Z 368.599,A -85,B 0,C 180,E1 19476.695,E2 19476.695} C_VEL
LIN {X 0,Y 568.345,Z 364.001,A -85,B 0,C 180,E1 19476.034,E2 19476.034} C_VEL
LIN {X 0,Y 564.582,Z 359.99,A -85,B 0,C 180,E1 19475.327,E2 19475.327} C_VEL
LIN {X 0,Y 562.996,Z 357.595,A -85,B 0,C 180,E1 19475.006,E2 19475.006} C_VEL
LIN {X 0,Y 559.847,Z 354.496,A -85,B 0,C 180,E1 19474.393,E2 19474.393} C_VEL
LIN {X 0,Y 558.221,Z 351.638,A -85,B 0,C 180,E1 19474.039,E2 19474.039} C_VEL
LIN {X 0,Y 555.311,Z 349.439,A -85,B 0,C 180,E1 19473.466,E2 19473.466} C_VEL
LIN {X 0,Y 553.74,Z 346.448,A -85,B 0,C 180,E1 19473.102,E2 19473.102} C_VEL
LIN {X 0,Y 553.504,Z 345.275,A -85,B 0,C 180,E1 19473.021,E2 19473.021} C_VEL
LIN {X 0,Y 553.467,Z 345.284,A -85,B 0,C 180,E1 19469.79,E2 19469.79} C_VEL
LIN {X 0,Y 553.47,Z 345.226,A -85,B 0,C 180,E1 19466.386,E2 19466.386} C_VEL
LIN {X 0,Y 553.504,Z 345.284,A -85,B 0,C 180,E1 19463.079,E2 19463.079} C_VEL
LIN {X 0,Y 553.446,Z 345.227,A -85,B 0,C 180,E1 19459.856,E2 19459.856} C_VEL
LIN {X 0,Y 553.502,Z 345.28,A -85,B 0,C 180,E1 19456.584,E2 19456.584} C_VEL
LIN {X 0,Y 553.446,Z 345.221,A -85,B 0,C 180,E1 19453.371,E2 19453.371} C_VEL
LIN {X 0,Y 553.457,Z 345.288,A -85,B 0,C 180,E1 19449.988,E2 19449.988} C_VEL
LIN {X 0,Y 553.476,Z 345.288,A -85,B 0,C 180,E1 19446.848,E2 19446.848} C_VEL
LIN {X 0,Y 553.435,Z 345.293,A -85,B 0,C 180,E1 19443.522,E2 19443.522} C_VEL
LIN {X 0,Y 553.505,Z 345.28,A -85,B 0,C 180,E1 19440.311,E2 19440.311} C_VEL
LIN {X 0,Y 553.429,Z 345.288,A -85,B 0,C 180,E1 19437.1,E2 19437.1} C_VEL
LIN {X 0,Y 553.447,Z 345.283,A -85,B 0,C 180,E1 19433.777,E2 19433.777} C_VEL
LIN {X 0,Y 553.425,Z 345.279,A -85,B 0,C 180,E1 19430.852,E2 19430.852} C_VEL
LIN {X 0,Y 553.42,Z 345.242,A -85,B 0,C 180,E1 19427.478,E2 19427.478} C_VEL
LIN {X 0,Y 553.432,Z 345.265,A -85,B 0,C 180,E1 19424.491,E2 19424.491} C_VEL
LIN {X 0,Y 553.407,Z 345.243,A -85,B 0,C 180,E1 19421.218,E2 19421.218} C_VEL
LIN {X 0,Y 553.463,Z 345.28,A -85,B 0,C 180,E1 19418.039,E2 19418.039} C_VEL
LIN {X 0,Y 553.396,Z 345.237,A -85,B 0,C 180,E1 19414.852,E2 19414.852} C_VEL
LIN {X 0,Y 553.456,Z 345.393,A -85,B 0,C 180,E1 19413.434,E2 19413.434} C_VEL
LIN {X 0,Y 554.866,Z 348.989,A -85,B 0,C 180,E1 19412.731,E2 19412.731} C_VEL
LIN {X 0,Y 557.312,Z 351.723,A -85,B 0,C 180,E1 19412.223,E2 19412.223} C_VEL
LIN {X 0,Y 560.799,Z 355.855,A -85,B 0,C 180,E1 19411.514,E2 19411.514} C_VEL
LIN {X 0,Y 564.888,Z 361.239,A -85,B 0,C 180,E1 19410.697,E2 19410.697} C_VEL
LIN {X 0,Y 566.63,Z 363.404,A -85,B 0,C 180,E1 19410.361,E2 19410.361} C_VEL
LIN {X 0,Y 577.981,Z 378.153,A -85,B 0,C 180,E1 19408.27,E2 19408.27} C_VEL
LIN {X 0,Y 592.058,Z 397.311,A -85,B 0,C 180,E1 19405.896,E2 19405.896} C_VEL
LIN {X 0,Y 609.388,Z 421.992,A -85,B 0,C 180,E1 19403.238,E2 19403.238} C_VEL
LIN {X 0,Y 614.056,Z 429.297,A -85,B 0,C 180,E1 19402.554,E2 19402.554} C_VEL
LIN {X 0,Y 607.523,Z 635.422,A -85,B 0,C 180,E1 19399.586,E2 19399.586} C_VEL
LIN {X 0,Y 601.512,Z 826.184,A -85,B 0,C 180,E1 19396.865,E2 19396.865} C_VEL
LIN {X 0,Y 600.051,Z 849.825,A -85,B 0,C 180,E1 19396.435,E2 19396.435} C_VEL
LIN {X 0,Y 597.619,Z 878.711,A -85,B 0,C 180,E1 19395.72,E2 19395.72} C_VEL
LIN {X 0,Y 595.342,Z 900.588,A -85,B 0,C 180,E1 19395.031,E2 19395.031} C_VEL
LIN {X 0,Y 592.958,Z 920.804,A -85,B 0,C 180,E1 19394.276,E2 19394.276} C_VEL
LIN {X 0,Y 590.459,Z 940.17,A -85,B 0,C 180,E1 19393.434,E2 19393.434} C_VEL
LIN {X 0,Y 587.711,Z 959.347,A -85,B 0,C 180,E1 19392.487,E2 19392.487} C_VEL
LIN {X 0,Y 584.554,Z 980.074,A -85,B 0,C 180,E1 19391.319,E2 19391.319} C_VEL
LIN {X 0,Y 580.382,Z 1005.819,A -85,B 0,C 180,E1 19389.637,E2 19389.637} C_VEL
LIN {X 0,Y 577.104,Z 1024.829,A -85,B 0,C 180,E1 19388.209,E2 19388.209} C_VEL
LIN {X 0,Y 574.033,Z 1042.217,A -85,B 0,C 180,E1 19386.749,E2 19386.749} C_VEL
LIN {X 0,Y 571.112,Z 1058.483,A -85,B 0,C 180,E1 19385.231,E2 19385.231} C_VEL
LIN {X 0,Y 568.193,Z 1074.809,A -85,B 0,C 180,E1 19383.543,E2 19383.543} C_VEL
LIN {X 0,Y 564.879,Z 1093.737,A -85,B 0,C 180,E1 19381.359,E2 19381.359} C_VEL
LIN {X 0,Y 561.878,Z 1111.058,A -85,B 0,C 180,E1 19379.066,E2 19379.066} C_VEL
LIN {X 0,Y 559.756,Z 1124.37,A -85,B 0,C 180,E1 19377.097,E2 19377.097} C_VEL
LIN {X 0,Y 557.749,Z 1137.625,A -85,B 0,C 180,E1 19374.916,E2 19374.916} C_VEL
LIN {X 0,Y 555.8,Z 1152.159,A -85,B 0,C 180,E1 19372.197,E2 19372.197} C_VEL
LIN {X 0,Y 554.442,Z 1163.603,A -85,B 0,C 180,E1 19369.709,E2 19369.709} C_VEL
LIN {X 0,Y 553.521,Z 1172.701,A -85,B 0,C 180,E1 19367.45,E2 19367.45} C_VEL
LIN {X 0,Y 552.863,Z 1180.919,A -85,B 0,C 180,E1 19365.096,E2 19365.096} C_VEL
LIN {X 0,Y 552.34,Z 1189.024,A -85,B 0,C 180,E1 19362.334,E2 19362.334} C_VEL
LIN {X 0,Y 552.078,Z 1195.293,A -85,B 0,C 180,E1 19359.592,E2 19359.592} C_VEL
LIN {X 0,Y 551.969,Z 1199.531,A -85,B 0,C 180,E1 19357.181,E2 19357.181} C_VEL
LIN {X 0,Y 551.918,Z 1202.668,A -85,B 0,C 180,E1 19354.677,E2 19354.677} C_VEL
LIN {X 0,Y 551.91,Z 1204.6,A -85,B 0,C 180,E1 19351.869,E2 19351.869} C_VEL
LIN {X 0,Y 551.895,Z 1204.872,A -85,B 0,C 180,E1 19349.378,E2 19349.378} C_VEL
LIN {X 0,Y 551.916,Z 1203.978,A -85,B 0,C 180,E1 19346.989,E2 19346.989} C_VEL
LIN {X 0,Y 551.93,Z 1201.873,A -85,B 0,C 180,E1 19344.595,E2 19344.595} C_VEL
LIN {X 0,Y 551.999,Z 1198.251,A -85,B 0,C 180,E1 19341.983,E2 19341.983} C_VEL
LIN {X 0,Y 552.169,Z 1192.609,A -85,B 0,C 180,E1 19339.145,E2 19339.145} C_VEL
LIN {X 0,Y 552.519,Z 1186.073,A -85,B 0,C 180,E1 19336.607,E2 19336.607} C_VEL
LIN {X 0,Y 552.999,Z 1178.801,A -85,B 0,C 180,E1 19334.264,E2 19334.264} C_VEL
LIN {X 0,Y 553.836,Z 1169.63,A -85,B 0,C 180,E1 19331.739,E2 19331.739} C_VEL
LIN {X 0,Y 555.152,Z 1157.326,A -85,B 0,C 180,E1 19328.887,E2 19328.887} C_VEL
LIN {X 0,Y 556.58,Z 1145.997,A -85,B 0,C 180,E1 19326.609,E2 19326.609} C_VEL
LIN {X 0,Y 558.32,Z 1133.823,A -85,B 0,C 180,E1 19324.432,E2 19324.432} C_VEL
LIN {X 0,Y 560.898,Z 1117.228,A -85,B 0,C 180,E1 19321.81,E2 19321.81} C_VEL
LIN {X 0,Y 563.604,Z 1100.916,A -85,B 0,C 180,E1 19319.566,E2 19319.566} C_VEL
LIN {X 0,Y 566.275,Z 1085.442,A -85,B 0,C 180,E1 19317.656,E2 19317.656} C_VEL
LIN {X 0,Y 569.654,Z 1066.709,A -85,B 0,C 180,E1 19315.585,E2 19315.585} C_VEL
LIN {X 0,Y 573.385,Z 1045.861,A -85,B 0,C 180,E1 19313.576,E2 19313.576} C_VEL
LIN {X 0,Y 576.465,Z 1028.465,A -85,B 0,C 180,E1 19312.084,E2 19312.084} C_VEL
LIN {X 0,Y 579.528,Z 1010.649,A -85,B 0,C 180,E1 19310.714,E2 19310.714} C_VEL
LIN {X 0,Y 582.646,Z 991.965,A -85,B 0,C 180,E1 19309.429,E2 19309.429} C_VEL
LIN {X 0,Y 586.145,Z 970.122,A -85,B 0,C 180,E1 19308.1,E2 19308.1} C_VEL
LIN {X 0,Y 589.847,Z 944.683,A -85,B 0,C 180,E1 19306.778,E2 19306.778} C_VEL
LIN {X 0,Y 592.628,Z 923.346,A -85,B 0,C 180,E1 19305.829,E2 19305.829} C_VEL
LIN {X 0,Y 595.083,Z 902.769,A -85,B 0,C 180,E1 19305.047,E2 19305.047} C_VEL
LIN {X 0,Y 597.279,Z 881.816,A -85,B 0,C 180,E1 19304.372,E2 19304.372} C_VEL
LIN {X 0,Y 599.357,Z 858.642,A -85,B 0,C 180,E1 19303.761,E2 19303.761} C_VEL
LIN {X 0,Y 601.348,Z 829.444,A -85,B 0,C 180,E1 19303.187,E2 19303.187} C_VEL
LIN {X 0,Y 603.423,Z 768.528,A -85,B 0,C 180,E1 19302.305,E2 19302.305} C_VEL
LIN {X 0,Y 610.644,Z 547.66,A -85,B 0,C 180,E1 19299.128,E2 19299.128} C_VEL
LIN {X 0,Y 614.743,Z 428.929,A -85,B 0,C 180,E1 19297.367,E2 19297.367} C_VEL
LIN {X 0,Y 604.515,Z 412.746,A -85,B 0,C 180,E1 19295.665,E2 19295.665} C_VEL
LIN {X 0,Y 594.303,Z 398.051,A -85,B 0,C 180,E1 19293.841,E2 19293.841} C_VEL
LIN {X 0,Y 583.949,Z 384.097,A -85,B 0,C 180,E1 19291.829,E2 19291.829} C_VEL
LIN {X 0,Y 575.34,Z 373.224,A -85,B 0,C 180,E1 19290.006,E2 19290.006} C_VEL
LIN {X 0,Y 571.601,Z 368.407,A -85,B 0,C 180,E1 19289.155,E2 19289.155} C_VEL
LIN {X 0,Y 567.859,Z 363.834,A -85,B 0,C 180,E1 19288.272,E2 19288.272} C_VEL
LIN {X 0,Y 566.315,Z 362.01,A -85,B 0,C 180,E1 19287.897,E2 19287.897} C_VEL
LIN {X 0,Y 562.846,Z 357.747,A -85,B 0,C 180,E1 19287.022,E2 19287.022} C_VEL
LIN {X 0,Y 557.892,Z 351.904,A -85,B 0,C 180,E1 19285.705,E2 19285.705} C_VEL
LIN {X 0,Y 554.495,Z 348.394,A -85,B 0,C 180,E1 19284.759,E2 19284.759} C_VEL
LIN {X 0,Y 553.47,Z 345.292,A -85,B 0,C 180,E1 19283.984,E2 19283.984} C_VEL
LIN {X 0,Y 553.401,Z 345.251,A -85,B 0,C 180,E1 19280.917,E2 19280.917} C_VEL
LIN {X 0,Y 553.439,Z 345.252,A -85,B 0,C 180,E1 19277.669,E2 19277.669} C_VEL
LIN {X 0,Y 553.403,Z 345.283,A -85,B 0,C 180,E1 19274.652,E2 19274.652} C_VEL
LIN {X 0,Y 553.411,Z 345.242,A -85,B 0,C 180,E1 19271.252,E2 19271.252} C_VEL
LIN {X 0,Y 553.43,Z 345.291,A -85,B 0,C 180,E1 19268.206,E2 19268.206} C_VEL
LIN {X 0,Y 553.407,Z 345.252,A -85,B 0,C 180,E1 19264.871,E2 19264.871} C_VEL
LIN {X 0,Y 553.468,Z 345.257,A -85,B 0,C 180,E1 19261.76,E2 19261.76} C_VEL
LIN {X 0,Y 553.413,Z 345.267,A -85,B 0,C 180,E1 19258.654,E2 19258.654} C_VEL
LIN {X 0,Y 553.476,Z 345.239,A -85,B 0,C 180,E1 19255.545,E2 19255.545} C_VEL
LIN {X 0,Y 553.421,Z 345.294,A -85,B 0,C 180,E1 19252.421,E2 19252.421} C_VEL
LIN {X 0,Y 553.484,Z 345.234,A -85,B 0,C 180,E1 19249.276,E2 19249.276} C_VEL
LIN {X 0,Y 553.427,Z 345.272,A -85,B 0,C 180,E1 19246.096,E2 19246.096} C_VEL
LIN {X 0,Y 553.472,Z 345.257,A -85,B 0,C 180,E1 19242.873,E2 19242.873} C_VEL
LIN {X 0,Y 553.49,Z 345.381,A -85,B 0,C 180,E1 19241.393,E2 19241.393} C_VEL
LIN {X 0,Y 554.44,Z 348.156,A -85,B 0,C 180,E1 19241.058,E2 19241.058} C_VEL
LIN {X 0,Y 556.651,Z 350.717,A -85,B 0,C 180,E1 19240.427,E2 19240.427} C_VEL
LIN {X 0,Y 559.106,Z 352.179,A -85,B 0,C 180,E1 19239.795,E2 19239.795} C_VEL
LIN {X 0,Y 561.182,Z 355.774,A -85,B 0,C 180,E1 19239.205,E2 19239.205} C_VEL
LIN {X 0,Y 564.61,Z 358.699,A -85,B 0,C 180,E1 19238.358,E2 19238.358} C_VEL
LIN {X 0,Y 567.193,Z 362.496,A -85,B 0,C 180,E1 19237.7,E2 19237.7} C_VEL
LIN {X 0,Y 569.993,Z 365.053,A -85,B 0,C 180,E1 19237.053,E2 19237.053} C_VEL
LIN {X 0,Y 573.042,Z 369.115,A -85,B 0,C 180,E1 19236.339,E2 19236.339} C_VEL
LIN {X 0,Y 575.25,Z 371.294,A -85,B 0,C 180,E1 19235.858,E2 19235.858} C_VEL
LIN {X 0,Y 578.86,Z 375.77,A -85,B 0,C 180,E1 19235.072,E2 19235.072} C_VEL
LIN {X 0,Y 580.775,Z 378.084,A -85,B 0,C 180,E1 19234.67,E2 19234.67} C_VEL
LIN {X 0,Y 585.661,Z 384.137,A -85,B 0,C 180,E1 19233.674,E2 19233.674} C_VEL
LIN {X 0,Y 592.048,Z 392.437,A -85,B 0,C 180,E1 19232.435,E2 19232.435} C_VEL
LIN {X 0,Y 601.985,Z 406.077,A -85,B 0,C 180,E1 19230.632,E2 19230.632} C_VEL
LIN {X 0,Y 612.967,Z 422.855,A -85,B 0,C 180,E1 19228.78,E2 19228.78} C_VEL
LIN {X 0,Y 614.805,Z 426.082,A -85,B 0,C 180,E1 19228.478,E2 19228.478} C_VEL
LIN {X 0,Y 607.111,Z 646.452,A -85,B 0,C 180,E1 19225.263,E2 19225.263} C_VEL
LIN {X 0,Y 601.529,Z 818,A -85,B 0,C 180,E1 19222.8,E2 19222.8} C_VEL
LIN {X 0,Y 601.479,Z 819.085,A -85,B 0,C 180,E1 19222.783,E2 19222.783} C_VEL
LIN {X 0,Y 600.121,Z 827.841,A -85,B 0,C 180,E1 19222.728,E2 19222.728} C_VEL
LIN {X 0,Y 594.838,Z 846.097,A -85,B 0,C 180,E1 19222.772,E2 19222.772} C_VEL
LIN {X 0,Y 593.552,Z 853.637,A -85,B 0,C 180,E1 19222.649,E2 19222.649} C_VEL
LIN {X 0,Y 591.528,Z 874.808,A -85,B 0,C 180,E1 19222.073,E2 19222.073} C_VEL
LIN {X 0,Y 589.233,Z 895.701,A -85,B 0,C 180,E1 19221.383,E2 19221.383} C_VEL
LIN {X 0,Y 586.311,Z 918.933,A -85,B 0,C 180,E1 19220.472,E2 19220.472} C_VEL
LIN {X 0,Y 582.429,Z 945.667,A -85,B 0,C 180,E1 19219.207,E2 19219.207} C_VEL
LIN {X 0,Y 579.203,Z 966.036,A -85,B 0,C 180,E1 19218.075,E2 19218.075} C_VEL
LIN {X 0,Y 575.848,Z 985.855,A -85,B 0,C 180,E1 19216.824,E2 19216.824} C_VEL
LIN {X 0,Y 572.007,Z 1007.425,A -85,B 0,C 180,E1 19215.28,E2 19215.28} C_VEL
LIN {X 0,Y 567.725,Z 1030.359,A -85,B 0,C 180,E1 19213.382,E2 19213.382} C_VEL
LIN {X 0,Y 564.333,Z 1048.206,A -85,B 0,C 180,E1 19211.705,E2 19211.705} C_VEL
LIN {X 0,Y 561.252,Z 1064.567,A -85,B 0,C 180,E1 19209.998,E2 19209.998} C_VEL
LIN {X 0,Y 557.885,Z 1082.87,A -85,B 0,C 180,E1 19207.868,E2 19207.868} C_VEL
LIN {X 0,Y 554.608,Z 1100.758,A -85,B 0,C 180,E1 19205.486,E2 19205.486} C_VEL
LIN {X 0,Y 552.235,Z 1114.712,A -85,B 0,C 180,E1 19203.395,E2 19203.395} C_VEL
LIN {X 0,Y 550.134,Z 1127.86,A -85,B 0,C 180,E1 19201.197,E2 19201.197} C_VEL
LIN {X 0,Y 548.051,Z 1142.412,A -85,B 0,C 180,E1 19198.431,E2 19198.431} C_VEL
LIN {X 0,Y 546.62,Z 1153.751,A -85,B 0,C 180,E1 19195.923,E2 19195.923} C_VEL
LIN {X 0,Y 545.624,Z 1162.901,A -85,B 0,C 180,E1 19193.611,E2 19193.611} C_VEL
LIN {X 0,Y 544.922,Z 1171.193,A -85,B 0,C 180,E1 19191.19,E2 19191.19} C_VEL
LIN {X 0,Y 544.349,Z 1179.557,A -85,B 0,C 180,E1 19188.257,E2 19188.257} C_VEL
LIN {X 0,Y 544.096,Z 1185.382,A -85,B 0,C 180,E1 19185.642,E2 19185.642} C_VEL
LIN {X 0,Y 543.974,Z 1189.466,A -85,B 0,C 180,E1 19183.283,E2 19183.283} C_VEL
LIN {X 0,Y 543.922,Z 1192.55,A -85,B 0,C 180,E1 19180.807,E2 19180.807} C_VEL
LIN {X 0,Y 543.913,Z 1194.56,A -85,B 0,C 180,E1 19178.031,E2 19178.031} C_VEL
LIN {X 0,Y 543.902,Z 1194.861,A -85,B 0,C 180,E1 19175.273,E2 19175.273} C_VEL
LIN {X 0,Y 543.91,Z 1194.009,A -85,B 0,C 180,E1 19172.95,E2 19172.95} C_VEL
LIN {X 0,Y 543.929,Z 1192.045,A -85,B 0,C 180,E1 19170.632,E2 19170.632} C_VEL
LIN {X 0,Y 543.981,Z 1188.839,A -85,B 0,C 180,E1 19168.209,E2 19168.209} C_VEL
LIN {X 0,Y 544.149,Z 1183.807,A -85,B 0,C 180,E1 19165.468,E2 19165.468} C_VEL
LIN {X 0,Y 544.523,Z 1176.777,A -85,B 0,C 180,E1 19162.615,E2 19162.615} C_VEL
LIN {X 0,Y 545.006,Z 1169.775,A -85,B 0,C 180,E1 19160.282,E2 19160.282} C_VEL
LIN {X 0,Y 545.733,Z 1161.979,A -85,B 0,C 180,E1 19158.051,E2 19158.051} C_VEL
LIN {X 0,Y 546.818,Z 1152.131,A -85,B 0,C 180,E1 19155.6,E2 19155.6} C_VEL
LIN {X 0,Y 548.553,Z 1138.579,A -85,B 0,C 180,E1 19152.716,E2 19152.716} C_VEL
LIN {X 0,Y 550.45,Z 1125.85,A -85,B 0,C 180,E1 19150.363,E2 19150.363} C_VEL
LIN {X 0,Y 552.58,Z 1112.529,A -85,B 0,C 180,E1 19148.168,E2 19148.168} C_VEL
LIN {X 0,Y 555.749,Z 1094.507,A -85,B 0,C 180,E1 19145.556,E2 19145.556} C_VEL
LIN {X 0,Y 558.665,Z 1078.324,A -85,B 0,C 180,E1 19143.495,E2 19143.495} C_VEL
LIN {X 0,Y 561.641,Z 1062.418,A -85,B 0,C 180,E1 19141.677,E2 19141.677} C_VEL
LIN {X 0,Y 565.046,Z 1044.448,A -85,B 0,C 180,E1 19139.831,E2 19139.831} C_VEL
LIN {X 0,Y 569.34,Z 1021.872,A -85,B 0,C 180,E1 19137.796,E2 19137.796} C_VEL
LIN {X 0,Y 572.843,Z 1002.772,A -85,B 0,C 180,E1 19136.285,E2 19136.285} C_VEL
LIN {X 0,Y 576.035,Z 984.791,A -85,B 0,C 180,E1 19135.016,E2 19135.016} C_VEL
LIN {X 0,Y 579.397,Z 964.875,A -85,B 0,C 180,E1 19133.768,E2 19133.768} C_VEL
LIN {X 0,Y 583.398,Z 939.721,A -85,B 0,C 180,E1 19132.4,E2 19132.4} C_VEL
LIN {X 0,Y 586.752,Z 915.318,A -85,B 0,C 180,E1 19131.288,E2 19131.288} C_VEL
LIN {X 0,Y 589.355,Z 894.625,A -85,B 0,C 180,E1 19130.49,E2 19130.49} C_VEL
LIN {X 0,Y 591.669,Z 873.505,A -85,B 0,C 180,E1 19129.8,E2 19129.8} C_VEL
LIN {X 0,Y 593.757,Z 851.096,A -85,B 0,C 180,E1 19129.198,E2 19129.198} C_VEL
LIN {X 0,Y 595.84,Z 822.6,A -85,B 0,C 180,E1 19128.619,E2 19128.619} C_VEL
LIN {X 0,Y 597.636,Z 774.18,A -85,B 0,C 180,E1 19127.906,E2 19127.906} C_VEL
LIN {X 0,Y 604.671,Z 555.252,A -85,B 0,C 180,E1 19124.773,E2 19124.773} C_VEL
LIN {X 0,Y 608.787,Z 429.563,A -85,B 0,C 180,E1 19122.938,E2 19122.938} C_VEL
LIN {X 0,Y 595.427,Z 410.431,A -85,B 0,C 180,E1 19120.914,E2 19120.914} C_VEL
LIN {X 0,Y 581.347,Z 391.064,A -85,B 0,C 180,E1 19118.603,E2 19118.603} C_VEL
LIN {X 0,Y 573.127,Z 380.689,A -85,B 0,C 180,E1 19117.163,E2 19117.163} C_VEL
LIN {X 0,Y 568.778,Z 375.282,A -85,B 0,C 180,E1 19116.364,E2 19116.364} C_VEL
LIN {X 0,Y 564.493,Z 370.034,A -85,B 0,C 180,E1 19115.552,E2 19115.552} C_VEL
LIN {X 0,Y 561.011,Z 365.697,A -85,B 0,C 180,E1 19114.867,E2 19114.867} C_VEL
LIN {X 0,Y 559.384,Z 363.969,A -85,B 0,C 180,E1 19114.547,E2 19114.547} C_VEL
LIN {X 0,Y 556.228,Z 360.026,A -85,B 0,C 180,E1 19113.898,E2 19113.898} C_VEL
LIN {X 0,Y 555.234,Z 358.698,A -85,B 0,C 180,E1 19113.688,E2 19113.688} C_VEL
LIN {X 0,Y 552.188,Z 355.769,A -85,B 0,C 180,E1 19113.059,E2 19113.059} C_VEL
LIN {X 0,Y 550.433,Z 352.671,A -85,B 0,C 180,E1 19112.651,E2 19112.651} C_VEL
LIN {X 0,Y 547.412,Z 350.519,A -85,B 0,C 180,E1 19112.017,E2 19112.017} C_VEL
LIN {X 0,Y 545.826,Z 347.602,A -85,B 0,C 180,E1 19111.627,E2 19111.627} C_VEL
LIN {X 0,Y 545.552,Z 346.272,A -85,B 0,C 180,E1 19111.52,E2 19111.52} C_VEL
LIN {X 0,Y 545.524,Z 346.245,A -85,B 0,C 180,E1 19108.162,E2 19108.162} C_VEL
LIN {X 0,Y 545.562,Z 346.235,A -85,B 0,C 180,E1 19104.816,E2 19104.816} C_VEL
LIN {X 0,Y 545.514,Z 346.228,A -85,B 0,C 180,E1 19101.618,E2 19101.618} C_VEL
LIN {X 0,Y 545.524,Z 346.256,A -85,B 0,C 180,E1 19098.155,E2 19098.155} C_VEL
LIN {X 0,Y 545.545,Z 346.217,A -85,B 0,C 180,E1 19094.977,E2 19094.977} C_VEL
LIN {X 0,Y 545.503,Z 346.246,A -85,B 0,C 180,E1 19091.739,E2 19091.739} C_VEL
LIN {X 0,Y 545.561,Z 346.258,A -85,B 0,C 180,E1 19088.431,E2 19088.431} C_VEL
LIN {X 0,Y 545.498,Z 346.263,A -85,B 0,C 180,E1 19085.259,E2 19085.259} C_VEL
LIN {X 0,Y 545.512,Z 346.263,A -85,B 0,C 180,E1 19081.891,E2 19081.891} C_VEL
LIN {X 0,Y 545.509,Z 346.27,A -85,B 0,C 180,E1 19078.845,E2 19078.845} C_VEL
LIN {X 0,Y 545.489,Z 346.274,A -85,B 0,C 180,E1 19075.479,E2 19075.479} C_VEL
LIN {X 0,Y 545.559,Z 346.266,A -85,B 0,C 180,E1 19072.205,E2 19072.205} C_VEL
LIN {X 0,Y 545.479,Z 346.28,A -85,B 0,C 180,E1 19069.01,E2 19069.01} C_VEL
LIN {X 0,Y 545.5,Z 346.218,A -85,B 0,C 180,E1 19065.673,E2 19065.673} C_VEL
LIN {X 0,Y 545.48,Z 346.272,A -85,B 0,C 180,E1 19062.615,E2 19062.615} C_VEL
LIN {X 0,Y 545.465,Z 346.233,A -85,B 0,C 180,E1 19059.168,E2 19059.168} C_VEL
LIN {X 0,Y 545.496,Z 346.239,A -85,B 0,C 180,E1 19056.157,E2 19056.157} C_VEL
LIN {X 0,Y 545.466,Z 346.297,A -85,B 0,C 180,E1 19054.832,E2 19054.832} C_VEL
LIN {X 0,Y 546.392,Z 349.07,A -85,B 0,C 180,E1 19054.326,E2 19054.326} C_VEL
LIN {X 0,Y 548.83,Z 351.759,A -85,B 0,C 180,E1 19053.781,E2 19053.781} C_VEL
LIN {X 0,Y 550.01,Z 353.083,A -85,B 0,C 180,E1 19053.522,E2 19053.522} C_VEL
LIN {X 0,Y 555.422,Z 359.856,A -85,B 0,C 180,E1 19052.354,E2 19052.354} C_VEL
LIN {X 0,Y 558.998,Z 364.221,A -85,B 0,C 180,E1 19051.618,E2 19051.618} C_VEL
LIN {X 0,Y 564.012,Z 370.631,A -85,B 0,C 180,E1 19050.618,E2 19050.618} C_VEL
LIN {X 0,Y 574.675,Z 384.518,A -85,B 0,C 180,E1 19048.622,E2 19048.622} C_VEL
LIN {X 0,Y 588.874,Z 404.077,A -85,B 0,C 180,E1 19046.185,E2 19046.185} C_VEL
LIN {X 0,Y 605.755,Z 428.274,A -85,B 0,C 180,E1 19043.556,E2 19043.556} C_VEL
LIN {X 0,Y 608.91,Z 433.285,A -85,B 0,C 180,E1 19043.085,E2 19043.085} C_VEL
LIN {X 0,Y 602.067,Z 641.129,A -85,B 0,C 180,E1 19040.079,E2 19040.079} C_VEL
LIN {X 0,Y 596.049,Z 825.812,A -85,B 0,C 180,E1 19037.432,E2 19037.432} C_VEL
LIN {X 0,Y 594.564,Z 849.025,A -85,B 0,C 180,E1 19037.011,E2 19037.011} C_VEL
LIN {X 0,Y 592.094,Z 877.662,A -85,B 0,C 180,E1 19036.308,E2 19036.308} C_VEL
LIN {X 0,Y 589.622,Z 900.464,A -85,B 0,C 180,E1 19035.59,E2 19035.59} C_VEL
LIN {X 0,Y 587.143,Z 920.685,A -85,B 0,C 180,E1 19034.832,E2 19034.832} C_VEL
LIN {X 0,Y 584.53,Z 940.056,A -85,B 0,C 180,E1 19033.987,E2 19033.987} C_VEL
LIN {X 0,Y 581.514,Z 960.244,A -85,B 0,C 180,E1 19032.981,E2 19032.981} C_VEL
LIN {X 0,Y 577.741,Z 984.104,A -85,B 0,C 180,E1 19031.612,E2 19031.612} C_VEL
LIN {X 0,Y 573.654,Z 1007.603,A -85,B 0,C 180,E1 19030.029,E2 19030.029} C_VEL
LIN {X 0,Y 570.317,Z 1026.066,A -85,B 0,C 180,E1 19028.619,E2 19028.619} C_VEL
LIN {X 0,Y 567.168,Z 1043.114,A -85,B 0,C 180,E1 19027.169,E2 19027.169} C_VEL
LIN {X 0,Y 564.041,Z 1059.817,A -85,B 0,C 180,E1 19025.59,E2 19025.59} C_VEL
LIN {X 0,Y 560.405,Z 1079.369,A -85,B 0,C 180,E1 19023.519,E2 19023.519} C_VEL
LIN {X 0,Y 556.886,Z 1097.973,A -85,B 0,C 180,E1 19021.258,E2 19021.258} C_VEL
LIN {X 0,Y 554.275,Z 1112.597,A -85,B 0,C 180,E1 19019.266,E2 19019.266} C_VEL
LIN {X 0,Y 551.95,Z 1126.469,A -85,B 0,C 180,E1 19017.162,E2 19017.162} C_VEL
LIN {X 0,Y 549.53,Z 1141.963,A -85,B 0,C 180,E1 19014.51,E2 19014.51} C_VEL
LIN {X 0,Y 547.732,Z 1154.761,A -85,B 0,C 180,E1 19011.972,E2 19011.972} C_VEL
LIN {X 0,Y 546.475,Z 1164.978,A -85,B 0,C 180,E1 19009.674,E2 19009.674} C_VEL
LIN {X 0,Y 545.488,Z 1174.403,A -85,B 0,C 180,E1 19007.252,E2 19007.252} C_VEL
LIN {X 0,Y 544.689,Z 1184.25,A -85,B 0,C 180,E1 19004.24,E2 19004.24} C_VEL
LIN {X 0,Y 544.27,Z 1191.078,A -85,B 0,C 180,E1 19001.659,E2 19001.659} C_VEL
LIN {X 0,Y 544.059,Z 1196.177,A -85,B 0,C 180,E1 18999.276,E2 18999.276} C_VEL
LIN {X 0,Y 543.955,Z 1200.485,A -85,B 0,C 180,E1 18996.65,E2 18996.65} C_VEL
LIN {X 0,Y 543.913,Z 1203.499,A -85,B 0,C 180,E1 18993.795,E2 18993.795} C_VEL
LIN {X 0,Y 543.913,Z 1204.713,A -85,B 0,C 180,E1 18991.37,E2 18991.37} C_VEL
LIN {X 0,Y 543.903,Z 1204.826,A -85,B 0,C 180,E1 18989.158,E2 18989.158} C_VEL
LIN {X 0,Y 543.917,Z 1203.907,A -85,B 0,C 180,E1 18986.839,E2 18986.839} C_VEL
LIN {X 0,Y 543.935,Z 1201.756,A -85,B 0,C 180,E1 18984.409,E2 18984.409} C_VEL
LIN {X 0,Y 544.012,Z 1197.908,A -85,B 0,C 180,E1 18981.652,E2 18981.652} C_VEL
LIN {X 0,Y 544.2,Z 1192.309,A -85,B 0,C 180,E1 18978.859,E2 18978.859} C_VEL
LIN {X 0,Y 544.568,Z 1186.07,A -85,B 0,C 180,E1 18976.408,E2 18976.408} C_VEL
LIN {X 0,Y 545.055,Z 1179.153,A -85,B 0,C 180,E1 18974.138,E2 18974.138} C_VEL
LIN {X 0,Y 545.869,Z 1170.679,A -85,B 0,C 180,E1 18971.747,E2 18971.747} C_VEL
LIN {X 0,Y 547.27,Z 1158.354,A -85,B 0,C 180,E1 18968.793,E2 18968.793} C_VEL
LIN {X 0,Y 548.838,Z 1146.568,A -85,B 0,C 180,E1 18966.373,E2 18966.373} C_VEL
LIN {X 0,Y 550.667,Z 1134.456,A -85,B 0,C 180,E1 18964.166,E2 18964.166} C_VEL
LIN {X 0,Y 553.261,Z 1118.749,A -85,B 0,C 180,E1 18961.621,E2 18961.621} C_VEL
LIN {X 0,Y 556.285,Z 1101.36,A -85,B 0,C 180,E1 18959.186,E2 18959.186} C_VEL
LIN {X 0,Y 559.019,Z 1086.366,A -85,B 0,C 180,E1 18957.306,E2 18957.306} C_VEL
LIN {X 0,Y 561.953,Z 1070.762,A -85,B 0,C 180,E1 18955.542,E2 18955.542} C_VEL
LIN {X 0,Y 565.77,Z 1050.835,A -85,B 0,C 180,E1 18953.526,E2 18953.526} C_VEL
LIN {X 0,Y 569.635,Z 1029.808,A -85,B 0,C 180,E1 18951.687,E2 18951.687} C_VEL
LIN {X 0,Y 572.848,Z 1012.008,A -85,B 0,C 180,E1 18950.296,E2 18950.296} C_VEL
LIN {X 0,Y 575.992,Z 994.044,A -85,B 0,C 180,E1 18949.038,E2 18949.038} C_VEL
LIN {X 0,Y 579.099,Z 975.421,A -85,B 0,C 180,E1 18947.873,E2 18947.873} C_VEL
LIN {X 0,Y 582.396,Z 954.44,A -85,B 0,C 180,E1 18946.715,E2 18946.715} C_VEL
LIN {X 0,Y 586.299,Z 927.205,A -85,B 0,C 180,E1 18945.438,E2 18945.438} C_VEL
LIN {X 0,Y 589.097,Z 904.855,A -85,B 0,C 180,E1 18944.567,E2 18944.567} C_VEL
LIN {X 0,Y 591.438,Z 883.606,A -85,B 0,C 180,E1 18943.869,E2 18943.869} C_VEL
LIN {X 0,Y 593.461,Z 862.373,A -85,B 0,C 180,E1 18943.294,E2 18943.294} C_VEL
LIN {X 0,Y 595.294,Z 839.002,A -85,B 0,C 180,E1 18942.791,E2 18942.791} C_VEL
LIN {X 0,Y 596.985,Z 802.866,A -85,B 0,C 180,E1 18942.223,E2 18942.223} C_VEL
LIN {X 0,Y 604.638,Z 578.254,A -85,B 0,C 180,E1 18938.977,E2 18938.977} C_VEL
LIN {X 0,Y 609.952,Z 433.144,A -85,B 0,C 180,E1 18936.825,E2 18936.825} C_VEL
LIN {X 0,Y 600.87,Z 418.635,A -85,B 0,C 180,E1 18935.27,E2 18935.27} C_VEL
LIN {X 0,Y 591.158,Z 404.49,A -85,B 0,C 180,E1 18933.495,E2 18933.495} C_VEL
LIN {X 0,Y 581.031,Z 390.753,A -85,B 0,C 180,E1 18931.486,E2 18931.486} C_VEL
LIN {X 0,Y 572.846,Z 380.263,A -85,B 0,C 180,E1 18929.717,E2 18929.717} C_VEL
LIN {X 0,Y 569.046,Z 375.395,A -85,B 0,C 180,E1 18928.838,E2 18928.838} C_VEL
LIN {X 0,Y 565.183,Z 370.428,A -85,B 0,C 180,E1 18927.901,E2 18927.901} C_VEL
LIN {X 0,Y 560.691,Z 365.072,A -85,B 0,C 180,E1 18926.762,E2 18926.762} C_VEL
LIN {X 0,Y 555.66,Z 358.977,A -85,B 0,C 180,E1 18925.395,E2 18925.395} C_VEL
LIN {X 0,Y 552.531,Z 355.812,A -85,B 0,C 180,E1 18924.511,E2 18924.511} C_VEL
LIN {X 0,Y 550.206,Z 352.605,A -85,B 0,C 180,E1 18923.794,E2 18923.794} C_VEL
LIN {X 0,Y 547.247,Z 350.369,A -85,B 0,C 180,E1 18922.903,E2 18922.903} C_VEL
LIN {X 0,Y 545.747,Z 347.377,A -85,B 0,C 180,E1 18922.288,E2 18922.288} C_VEL
LIN {X 0,Y 545.528,Z 346.227,A -85,B 0,C 180,E1 18921.957,E2 18921.957} C_VEL
LIN {X 0,Y 545.468,Z 346.281,A -85,B 0,C 180,E1 18918.822,E2 18918.822} C_VEL
LIN {X 0,Y 545.477,Z 346.243,A -85,B 0,C 180,E1 18915.414,E2 18915.414} C_VEL
LIN {X 0,Y 545.469,Z 346.244,A -85,B 0,C 180,E1 18912.492,E2 18912.492} C_VEL
LIN {X 0,Y 545.469,Z 346.277,A -85,B 0,C 180,E1 18909.07,E2 18909.07} C_VEL
LIN {X 0,Y 545.494,Z 346.227,A -85,B 0,C 180,E1 18906.103,E2 18906.103} C_VEL
LIN {X 0,Y 545.476,Z 346.284,A -85,B 0,C 180,E1 18902.837,E2 18902.837} C_VEL
LIN {X 0,Y 545.551,Z 346.222,A -85,B 0,C 180,E1 18899.58,E2 18899.58} C_VEL
LIN {X 0,Y 545.475,Z 346.252,A -85,B 0,C 180,E1 18896.322,E2 18896.322} C_VEL
LIN {X 0,Y 545.505,Z 346.258,A -85,B 0,C 180,E1 18892.946,E2 18892.946} C_VEL
LIN {X 0,Y 545.497,Z 346.229,A -85,B 0,C 180,E1 18889.865,E2 18889.865} C_VEL
LIN {X 0,Y 545.496,Z 346.276,A -85,B 0,C 180,E1 18886.539,E2 18886.539} C_VEL
LIN {X 0,Y 545.533,Z 346.314,A -85,B 0,C 180,E1 18883.535,E2 18883.535} C_VEL
LIN {X 0,Y 546.447,Z 349.036,A -85,B 0,C 180,E1 18883.168,E2 18883.168} C_VEL
LIN {X 0,Y 548.677,Z 351.707,A -85,B 0,C 180,E1 18882.446,E2 18882.446} C_VEL
LIN {X 0,Y 551.324,Z 353.165,A -85,B 0,C 180,E1 18881.687,E2 18881.687} C_VEL
LIN {X 0,Y 553.253,Z 356.714,A -85,B 0,C 180,E1 18881.07,E2 18881.07} C_VEL
LIN {X 0,Y 556.258,Z 359.181,A -85,B 0,C 180,E1 18880.249,E2 18880.249} C_VEL
LIN {X 0,Y 557.065,Z 359.899,A -85,B 0,C 180,E1 18880.033,E2 18880.033} C_VEL
LIN {X 0,Y 559.742,Z 363.818,A -85,B 0,C 180,E1 18879.286,E2 18879.286} C_VEL
LIN {X 0,Y 562.477,Z 366.237,A -85,B 0,C 180,E1 18878.601,E2 18878.601} C_VEL
LIN {X 0,Y 565.54,Z 370.318,A -85,B 0,C 180,E1 18877.823,E2 18877.823} C_VEL
LIN {X 0,Y 567.807,Z 372.546,A -85,B 0,C 180,E1 18877.288,E2 18877.288} C_VEL
LIN {X 0,Y 571.255,Z 376.841,A -85,B 0,C 180,E1 18876.479,E2 18876.479} C_VEL
LIN {X 0,Y 572.994,Z 378.734,A -85,B 0,C 180,E1 18876.091,E2 18876.091} C_VEL
LIN {X 0,Y 576.824,Z 383.301,A -85,B 0,C 180,E1 18875.252,E2 18875.252} C_VEL
LIN {X 0,Y 583.338,Z 391.559,A -85,B 0,C 180,E1 18873.89,E2 18873.89} C_VEL
LIN {X 0,Y 589.331,Z 399.45,A -85,B 0,C 180,E1 18872.708,E2 18872.708} C_VEL
LIN {X 0,Y 599.163,Z 413.149,A -85,B 0,C 180,E1 18870.892,E2 18870.892} C_VEL
LIN {X 0,Y 609.676,Z 429.426,A -85,B 0,C 180,E1 18869.084,E2 18869.084} C_VEL
LIN {X 0,Y 609.957,Z 430.454,A -85,B 0,C 180,E1 18869.026,E2 18869.026} C_VEL
LIN {X 0,Y 601.911,Z 649.537,A -85,B 0,C 180,E1 18865.807,E2 18865.807} C_VEL
LIN {X 0,Y 596.095,Z 817.919,A -85,B 0,C 180,E1 18863.367,E2 18863.367} C_VEL
LIN {X 0,Y 594.479,Z 842.907,A -85,B 0,C 180,E1 18862.901,E2 18862.901} C_VEL
LIN {X 0,Y 593.552,Z 853.637,A -85,B 0,C 180,E1 18862.649,E2 18862.649} C_VEL
LIN {X 0,Y 592.155,Z 861.186,A -85,B 0,C 180,E1 18862.538,E2 18862.538} C_VEL
LIN {X 0,Y 585.868,Z 881.402,A -85,B 0,C 180,E1 18862.394,E2 18862.394} C_VEL
LIN {X 0,Y 584.576,Z 887.696,A -85,B 0,C 180,E1 18862.237,E2 18862.237} C_VEL
LIN {X 0,Y 581.701,Z 910.31,A -85,B 0,C 180,E1 18861.394,E2 18861.394} C_VEL
LIN {X 0,Y 578.912,Z 930.026,A -85,B 0,C 180,E1 18860.535,E2 18860.535} C_VEL
LIN {X 0,Y 575.748,Z 950.301,A -85,B 0,C 180,E1 18859.521,E2 18859.521} C_VEL
LIN {X 0,Y 572.111,Z 972.086,A -85,B 0,C 180,E1 18858.267,E2 18858.267} C_VEL
LIN {X 0,Y 567.642,Z 996.816,A -85,B 0,C 180,E1 18856.608,E2 18856.608} C_VEL
LIN {X 0,Y 563.927,Z 1016.197,A -85,B 0,C 180,E1 18855.114,E2 18855.114} C_VEL
LIN {X 0,Y 560.457,Z 1033.858,A -85,B 0,C 180,E1 18853.587,E2 18853.587} C_VEL
LIN {X 0,Y 556.977,Z 1051.344,A -85,B 0,C 180,E1 18851.897,E2 18851.897} C_VEL
LIN {X 0,Y 552.92,Z 1071.816,A -85,B 0,C 180,E1 18849.668,E2 18849.668} C_VEL
LIN {X 0,Y 549.46,Z 1089.295,A -85,B 0,C 180,E1 18847.493,E2 18847.493} C_VEL
LIN {X 0,Y 546.831,Z 1103.349,A -85,B 0,C 180,E1 18845.541,E2 18845.541} C_VEL
LIN {X 0,Y 544.284,Z 1117.732,A -85,B 0,C 180,E1 18843.317,E2 18843.317} C_VEL
LIN {X 0,Y 541.596,Z 1134.004,A -85,B 0,C 180,E1 18840.438,E2 18840.438} C_VEL
LIN {X 0,Y 539.879,Z 1145.68,A -85,B 0,C 180,E1 18838.061,E2 18838.061} C_VEL
LIN {X 0,Y 538.581,Z 1155.715,A -85,B 0,C 180,E1 18835.748,E2 18835.748} C_VEL
LIN {X 0,Y 537.43,Z 1166.498,A -85,B 0,C 180,E1 18832.882,E2 18832.882} C_VEL
LIN {X 0,Y 536.68,Z 1175.068,A -85,B 0,C 180,E1 18830.114,E2 18830.114} C_VEL
LIN {X 0,Y 536.294,Z 1181.318,A -85,B 0,C 180,E1 18827.686,E2 18827.686} C_VEL
LIN {X 0,Y 536.066,Z 1186.408,A -85,B 0,C 180,E1 18825.247,E2 18825.247} C_VEL
LIN {X 0,Y 535.951,Z 1190.768,A -85,B 0,C 180,E1 18822.498,E2 18822.498} C_VEL
LIN {X 0,Y 535.915,Z 1193.586,A -85,B 0,C 180,E1 18819.666,E2 18819.666} C_VEL
LIN {X 0,Y 535.914,Z 1194.725,A -85,B 0,C 180,E1 18817.288,E2 18817.288} C_VEL
LIN {X 0,Y 535.903,Z 1194.812,A -85,B 0,C 180,E1 18815.03,E2 18815.03} C_VEL
LIN {X 0,Y 535.911,Z 1193.927,A -85,B 0,C 180,E1 18812.78,E2 18812.78} C_VEL
LIN {X 0,Y 535.939,Z 1191.797,A -85,B 0,C 180,E1 18810.32,E2 18810.32} C_VEL
LIN {X 0,Y 536.02,Z 1188.005,A -85,B 0,C 180,E1 18807.541,E2 18807.541} C_VEL
LIN {X 0,Y 536.231,Z 1182.312,A -85,B 0,C 180,E1 18804.65,E2 18804.65} C_VEL
LIN {X 0,Y 536.611,Z 1176.135,A -85,B 0,C 180,E1 18802.182,E2 18802.182} C_VEL
LIN {X 0,Y 537.169,Z 1169.033,A -85,B 0,C 180,E1 18799.814,E2 18799.814} C_VEL
LIN {X 0,Y 538.107,Z 1159.945,A -85,B 0,C 180,E1 18797.225,E2 18797.225} C_VEL
LIN {X 0,Y 539.594,Z 1147.766,A -85,B 0,C 180,E1 18794.303,E2 18794.303} C_VEL
LIN {X 0,Y 541.235,Z 1136.284,A -85,B 0,C 180,E1 18791.919,E2 18791.919} C_VEL
LIN {X 0,Y 543.197,Z 1123.932,A -85,B 0,C 180,E1 18789.641,E2 18789.641} C_VEL
LIN {X 0,Y 546.162,Z 1107.217,A -85,B 0,C 180,E1 18786.935,E2 18786.935} C_VEL
LIN {X 0,Y 548.95,Z 1091.97,A -85,B 0,C 180,E1 18784.772,E2 18784.772} C_VEL
LIN {X 0,Y 551.896,Z 1076.739,A -85,B 0,C 180,E1 18782.835,E2 18782.835} C_VEL
LIN {X 0,Y 555.26,Z 1059.888,A -85,B 0,C 180,E1 18780.909,E2 18780.909} C_VEL
LIN {X 0,Y 559.716,Z 1037.716,A -85,B 0,C 180,E1 18778.678,E2 18778.678} C_VEL
LIN {X 0,Y 563.317,Z 1019.39,A -85,B 0,C 180,E1 18777.061,E2 18777.061} C_VEL
LIN {X 0,Y 566.799,Z 1001.252,A -85,B 0,C 180,E1 18775.632,E2 18775.632} C_VEL
LIN {X 0,Y 570.214,Z 982.785,A -85,B 0,C 180,E1 18774.335,E2 18774.335} C_VEL
LIN {X 0,Y 574.008,Z 961.234,A -85,B 0,C 180,E1 18772.998,E2 18772.998} C_VEL
LIN {X 0,Y 578.015,Z 936.251,A -85,B 0,C 180,E1 18771.673,E2 18771.673} C_VEL
LIN {X 0,Y 581.043,Z 914.978,A -85,B 0,C 180,E1 18770.708,E2 18770.708} C_VEL
LIN {X 0,Y 583.751,Z 894.213,A -85,B 0,C 180,E1 18769.907,E2 18769.907} C_VEL
LIN {X 0,Y 586.121,Z 873.35,A -85,B 0,C 180,E1 18769.225,E2 18769.225} C_VEL
LIN {X 0,Y 588.241,Z 851.26,A -85,B 0,C 180,E1 18768.632,E2 18768.632} C_VEL
LIN {X 0,Y 590.385,Z 822.886,A -85,B 0,C 180,E1 18768.053,E2 18768.053} C_VEL
LIN {X 0,Y 592.221,Z 774.859,A -85,B 0,C 180,E1 18767.343,E2 18767.343} C_VEL
LIN {X 0,Y 599.527,Z 555.573,A -85,B 0,C 180,E1 18764.189,E2 18764.189} C_VEL
LIN {X 0,Y 603.766,Z 433.752,A -85,B 0,C 180,E1 18762.412,E2 18762.412} C_VEL
LIN {X 0,Y 590.734,Z 415.171,A -85,B 0,C 180,E1 18760.394,E2 18760.394} C_VEL
LIN {X 0,Y 578.159,Z 397.668,A -85,B 0,C 180,E1 18758.285,E2 18758.285} C_VEL
LIN {X 0,Y 569.89,Z 387.179,A -85,B 0,C 180,E1 18756.811,E2 18756.811} C_VEL
LIN {X 0,Y 565.332,Z 381.516,A -85,B 0,C 180,E1 18755.959,E2 18755.959} C_VEL
LIN {X 0,Y 561.576,Z 376.858,A -85,B 0,C 180,E1 18755.232,E2 18755.232} C_VEL
LIN {X 0,Y 557.112,Z 371.362,A -85,B 0,C 180,E1 18754.337,E2 18754.337} C_VEL
LIN {X 0,Y 553.616,Z 367.163,A -85,B 0,C 180,E1 18753.613,E2 18753.613} C_VEL
LIN {X 0,Y 552.285,Z 365.599,A -85,B 0,C 180,E1 18753.331,E2 18753.331} C_VEL
LIN {X 0,Y 549.096,Z 362.051,A -85,B 0,C 180,E1 18752.647,E2 18752.647} C_VEL
LIN {X 0,Y 547.746,Z 359.931,A -85,B 0,C 180,E1 18752.335,E2 18752.335} C_VEL
LIN {X 0,Y 544.587,Z 357.169,A -85,B 0,C 180,E1 18751.645,E2 18751.645} C_VEL
LIN {X 0,Y 542.728,Z 353.744,A -85,B 0,C 180,E1 18751.178,E2 18751.178} C_VEL
LIN {X 0,Y 539.525,Z 351.538,A -85,B 0,C 180,E1 18750.456,E2 18750.456} C_VEL
LIN {X 0,Y 537.918,Z 348.752,A -85,B 0,C 180,E1 18750.034,E2 18750.034} C_VEL
LIN {X 0,Y 537.587,Z 347.259,A -85,B 0,C 180,E1 18749.899,E2 18749.899} C_VEL
LIN {X 0,Y 537.601,Z 347.198,A -85,B 0,C 180,E1 18746.512,E2 18746.512} C_VEL
LIN {X 0,Y 537.624,Z 347.261,A -85,B 0,C 180,E1 18743.106,E2 18743.106} C_VEL
LIN {X 0,Y 537.568,Z 347.201,A -85,B 0,C 180,E1 18739.752,E2 18739.752} C_VEL
LIN {X 0,Y 537.61,Z 347.256,A -85,B 0,C 180,E1 18736.422,E2 18736.422} C_VEL
LIN {X 0,Y 537.575,Z 347.194,A -85,B 0,C 180,E1 18733.225,E2 18733.225} C_VEL
LIN {X 0,Y 537.571,Z 347.265,A -85,B 0,C 180,E1 18729.853,E2 18729.853} C_VEL
LIN {X 0,Y 537.63,Z 347.261,A -85,B 0,C 180,E1 18726.514,E2 18726.514} C_VEL
LIN {X 0,Y 537.561,Z 347.27,A -85,B 0,C 180,E1 18723.199,E2 18723.199} C_VEL
LIN {X 0,Y 537.568,Z 347.27,A -85,B 0,C 180,E1 18719.787,E2 18719.787} C_VEL
LIN {X 0,Y 537.589,Z 347.265,A -85,B 0,C 180,E1 18716.588,E2 18716.588} C_VEL
LIN {X 0,Y 537.545,Z 347.272,A -85,B 0,C 180,E1 18713.27,E2 18713.27} C_VEL
LIN {X 0,Y 537.603,Z 347.261,A -85,B 0,C 180,E1 18710.039,E2 18710.039} C_VEL
LIN {X 0,Y 537.536,Z 347.204,A -85,B 0,C 180,E1 18706.774,E2 18706.774} C_VEL
LIN {X 0,Y 537.54,Z 347.275,A -85,B 0,C 180,E1 18703.326,E2 18703.326} C_VEL
LIN {X 0,Y 537.577,Z 347.201,A -85,B 0,C 180,E1 18700.1,E2 18700.1} C_VEL
LIN {X 0,Y 537.521,Z 347.257,A -85,B 0,C 180,E1 18696.89,E2 18696.89} C_VEL
LIN {X 0,Y 537.55,Z 347.293,A -85,B 0,C 180,E1 18696.31,E2 18696.31} C_VEL
LIN {X 0,Y 537.993,Z 348.978,A -85,B 0,C 180,E1 18696.047,E2 18696.047} C_VEL
LIN {X 0,Y 539.934,Z 351.972,A -85,B 0,C 180,E1 18695.55,E2 18695.55} C_VEL
LIN {X 0,Y 542.561,Z 354.092,A -85,B 0,C 180,E1 18694.95,E2 18694.95} C_VEL
LIN {X 0,Y 545.713,Z 358.39,A -85,B 0,C 180,E1 18694.204,E2 18694.204} C_VEL
LIN {X 0,Y 547.531,Z 360.267,A -85,B 0,C 180,E1 18693.802,E2 18693.802} C_VEL
LIN {X 0,Y 556.216,Z 371.098,A -85,B 0,C 180,E1 18691.931,E2 18691.931} C_VEL
LIN {X 0,Y 561.518,Z 377.99,A -85,B 0,C 180,E1 18690.855,E2 18690.855} C_VEL
LIN {X 0,Y 571.507,Z 391.067,A -85,B 0,C 180,E1 18688.957,E2 18688.957} C_VEL
LIN {X 0,Y 585.579,Z 410.64,A -85,B 0,C 180,E1 18686.498,E2 18686.498} C_VEL
LIN {X 0,Y 602.135,Z 434.555,A -85,B 0,C 180,E1 18683.878,E2 18683.878} C_VEL
LIN {X 0,Y 603.799,Z 437.378,A -85,B 0,C 180,E1 18683.621,E2 18683.621} C_VEL
LIN {X 0,Y 596.63,Z 646.77,A -85,B 0,C 180,E1 18680.579,E2 18680.579} C_VEL
LIN {X 0,Y 590.59,Z 825.973,A -85,B 0,C 180,E1 18677.999,E2 18677.999} C_VEL
LIN {X 0,Y 589.021,Z 849.708,A -85,B 0,C 180,E1 18677.566,E2 18677.566} C_VEL
LIN {X 0,Y 586.416,Z 878.535,A -85,B 0,C 180,E1 18676.849,E2 18676.849} C_VEL
LIN {X 0,Y 583.873,Z 901.081,A -85,B 0,C 180,E1 18676.134,E2 18676.134} C_VEL
LIN {X 0,Y 581.389,Z 920.565,A -85,B 0,C 180,E1 18675.398,E2 18675.398} C_VEL
LIN {X 0,Y 578.655,Z 939.939,A -85,B 0,C 180,E1 18674.551,E2 18674.551} C_VEL
LIN {X 0,Y 575.531,Z 960.03,A -85,B 0,C 180,E1 18673.546,E2 18673.546} C_VEL
LIN {X 0,Y 571.655,Z 983.471,A -85,B 0,C 180,E1 18672.195,E2 18672.195} C_VEL
LIN {X 0,Y 567.443,Z 1006.76,A -85,B 0,C 180,E1 18670.624,E2 18670.624} C_VEL
LIN {X 0,Y 563.961,Z 1025.178,A -85,B 0,C 180,E1 18669.214,E2 18669.214} C_VEL
LIN {X 0,Y 560.572,Z 1042.648,A -85,B 0,C 180,E1 18667.72,E2 18667.72} C_VEL
LIN {X 0,Y 557.271,Z 1059.51,A -85,B 0,C 180,E1 18666.115,E2 18666.115} C_VEL
LIN {X 0,Y 553.706,Z 1077.847,A -85,B 0,C 180,E1 18664.167,E2 18664.167} C_VEL
LIN {X 0,Y 549.902,Z 1097.125,A -85,B 0,C 180,E1 18661.824,E2 18661.824} C_VEL
LIN {X 0,Y 547.092,Z 1111.825,A -85,B 0,C 180,E1 18659.81,E2 18659.81} C_VEL
LIN {X 0,Y 544.705,Z 1125.166,A -85,B 0,C 180,E1 18657.774,E2 18657.774} C_VEL
LIN {X 0,Y 542.305,Z 1139.526,A -85,B 0,C 180,E1 18655.325,E2 18655.325} C_VEL
LIN {X 0,Y 540.147,Z 1153.748,A -85,B 0,C 180,E1 18652.523,E2 18652.523} C_VEL
LIN {X 0,Y 538.779,Z 1164.059,A -85,B 0,C 180,E1 18650.193,E2 18650.193} C_VEL
LIN {X 0,Y 537.745,Z 1173.104,A -85,B 0,C 180,E1 18647.867,E2 18647.867} C_VEL
LIN {X 0,Y 536.937,Z 1181.977,A -85,B 0,C 180,E1 18645.223,E2 18645.223} C_VEL
LIN {X 0,Y 536.35,Z 1190.058,A -85,B 0,C 180,E1 18642.271,E2 18642.271} C_VEL
LIN {X 0,Y 536.098,Z 1195.494,A -85,B 0,C 180,E1 18639.772,E2 18639.772} C_VEL
LIN {X 0,Y 535.98,Z 1199.526,A -85,B 0,C 180,E1 18637.396,E2 18637.396} C_VEL
LIN {X 0,Y 535.924,Z 1202.549,A -85,B 0,C 180,E1 18634.924,E2 18634.924} C_VEL
LIN {X 0,Y 535.912,Z 1204.577,A -85,B 0,C 180,E1 18632.032,E2 18632.032} C_VEL
LIN {X 0,Y 535.895,Z 1204.872,A -85,B 0,C 180,E1 18629.359,E2 18629.359} C_VEL
LIN {X 0,Y 535.915,Z 1204.041,A -85,B 0,C 180,E1 18627.006,E2 18627.006} C_VEL
LIN {X 0,Y 535.931,Z 1202.094,A -85,B 0,C 180,E1 18624.648,E2 18624.648} C_VEL
LIN {X 0,Y 535.986,Z 1199.047,A -85,B 0,C 180,E1 18622.281,E2 18622.281} C_VEL
LIN {X 0,Y 536.153,Z 1194.256,A -85,B 0,C 180,E1 18619.578,E2 18619.578} C_VEL
LIN {X 0,Y 536.548,Z 1187.176,A -85,B 0,C 180,E1 18616.602,E2 18616.602} C_VEL
LIN {X 0,Y 537.084,Z 1179.859,A -85,B 0,C 180,E1 18614.118,E2 18614.118} C_VEL
LIN {X 0,Y 537.886,Z 1171.844,A -85,B 0,C 180,E1 18611.79,E2 18611.79} C_VEL
LIN {X 0,Y 539.073,Z 1161.773,A -85,B 0,C 180,E1 18609.252,E2 18609.252} C_VEL
LIN {X 0,Y 540.935,Z 1148.287,A -85,B 0,C 180,E1 18606.353,E2 18606.353} C_VEL
LIN {X 0,Y 542.817,Z 1136.359,A -85,B 0,C 180,E1 18604.116,E2 18604.116} C_VEL
LIN {X 0,Y 545.002,Z 1123.401,A -85,B 0,C 180,E1 18601.942,E2 18601.942} C_VEL
LIN {X 0,Y 548.026,Z 1107.205,A -85,B 0,C 180,E1 18599.522,E2 18599.522} C_VEL
LIN {X 0,Y 551.437,Z 1089.142,A -85,B 0,C 180,E1 18597.17,E2 18597.17} C_VEL
LIN {X 0,Y 554.457,Z 1073.795,A -85,B 0,C 180,E1 18595.386,E2 18595.386} C_VEL
LIN {X 0,Y 557.689,Z 1057.278,A -85,B 0,C 180,E1 18593.662,E2 18593.662} C_VEL
LIN {X 0,Y 561.306,Z 1038.863,A -85,B 0,C 180,E1 18591.94,E2 18591.94} C_VEL
LIN {X 0,Y 565.93,Z 1014.844,A -85,B 0,C 180,E1 18589.977,E2 18589.977} C_VEL
LIN {X 0,Y 569.423,Z 995.8,A -85,B 0,C 180,E1 18588.616,E2 18588.616} C_VEL
LIN {X 0,Y 572.677,Z 977.196,A -85,B 0,C 180,E1 18587.432,E2 18587.432} C_VEL
LIN {X 0,Y 575.823,Z 958.07,A -85,B 0,C 180,E1 18586.352,E2 18586.352} C_VEL
LIN {X 0,Y 578.974,Z 937.614,A -85,B 0,C 180,E1 18585.342,E2 18585.342} C_VEL
LIN {X 0,Y 582.551,Z 912.132,A -85,B 0,C 180,E1 18584.263,E2 18584.263} C_VEL
LIN {X 0,Y 585.632,Z 885.811,A -85,B 0,C 180,E1 18583.365,E2 18583.365} C_VEL
LIN {X 0,Y 587.816,Z 864.324,A -85,B 0,C 180,E1 18582.768,E2 18582.768} C_VEL
LIN {X 0,Y 589.595,Z 843.05,A -85,B 0,C 180,E1 18582.293,E2 18582.293} C_VEL
LIN {X 0,Y 591.034,Z 819.59,A -85,B 0,C 180,E1 18581.889,E2 18581.889} C_VEL
LIN {X 0,Y 599.03,Z 597.419,A -85,B 0,C 180,E1 18578.65,E2 18578.65} C_VEL
LIN {X 0,Y 605.184,Z 437.163,A -85,B 0,C 180,E1 18576.263,E2 18576.263} C_VEL
LIN {X 0,Y 594.91,Z 420.934,A -85,B 0,C 180,E1 18574.442,E2 18574.442} C_VEL
LIN {X 0,Y 585.986,Z 408.124,A -85,B 0,C 180,E1 18572.746,E2 18572.746} C_VEL
LIN {X 0,Y 577.387,Z 396.466,A -85,B 0,C 180,E1 18570.982,E2 18570.982} C_VEL
LIN {X 0,Y 570.574,Z 387.536,A -85,B 0,C 180,E1 18569.472,E2 18569.472} C_VEL
LIN {X 0,Y 566.513,Z 382.365,A -85,B 0,C 180,E1 18568.518,E2 18568.518} C_VEL
LIN {X 0,Y 561.753,Z 376.383,A -85,B 0,C 180,E1 18567.337,E2 18567.337} C_VEL
LIN {X 0,Y 556.844,Z 370.373,A -85,B 0,C 180,E1 18566.042,E2 18566.042} C_VEL
LIN {X 0,Y 553.022,Z 365.867,A -85,B 0,C 180,E1 18564.972,E2 18564.972} C_VEL
LIN {X 0,Y 549.78,Z 362.087,A -85,B 0,C 180,E1 18564.013,E2 18564.013} C_VEL
LIN {X 0,Y 548.267,Z 360.162,A -85,B 0,C 180,E1 18563.541,E2 18563.541} C_VEL
LIN {X 0,Y 545.218,Z 357.551,A -85,B 0,C 180,E1 18562.595,E2 18562.595} C_VEL
LIN {X 0,Y 543.108,Z 353.858,A -85,B 0,C 180,E1 18561.832,E2 18561.832} C_VEL
LIN {X 0,Y 539.938,Z 352.019,A -85,B 0,C 180,E1 18560.771,E2 18560.771} C_VEL
LIN {X 0,Y 538.109,Z 349.229,A -85,B 0,C 180,E1 18560.049,E2 18560.049} C_VEL
LIN {X 0,Y 537.568,Z 347.251,A -85,B 0,C 180,E1 18559.721,E2 18559.721} C_VEL
LIN {X 0,Y 537.532,Z 347.217,A -85,B 0,C 180,E1 18556.535,E2 18556.535} C_VEL
LIN {X 0,Y 537.526,Z 347.251,A -85,B 0,C 180,E1 18553.117,E2 18553.117} C_VEL
LIN {X 0,Y 537.588,Z 347.229,A -85,B 0,C 180,E1 18549.853,E2 18549.853} C_VEL
LIN {X 0,Y 537.523,Z 347.223,A -85,B 0,C 180,E1 18546.631,E2 18546.631} C_VEL
LIN {X 0,Y 537.569,Z 347.268,A -85,B 0,C 180,E1 18543.306,E2 18543.306} C_VEL
LIN {X 0,Y 537.541,Z 347.213,A -85,B 0,C 180,E1 18540.213,E2 18540.213} C_VEL
LIN {X 0,Y 537.546,Z 347.255,A -85,B 0,C 180,E1 18536.801,E2 18536.801} C_VEL
LIN {X 0,Y 537.607,Z 347.222,A -85,B 0,C 180,E1 18533.486,E2 18533.486} C_VEL
LIN {X 0,Y 537.541,Z 347.223,A -85,B 0,C 180,E1 18530.255,E2 18530.255} C_VEL
LIN {X 0,Y 537.584,Z 347.269,A -85,B 0,C 180,E1 18526.884,E2 18526.884} C_VEL
LIN {X 0,Y 537.575,Z 347.407,A -85,B 0,C 180,E1 18526.007,E2 18526.007} C_VEL
LIN {X 0,Y 538.466,Z 350.013,A -85,B 0,C 180,E1 18525.592,E2 18525.592} C_VEL
LIN {X 0,Y 541.086,Z 352.898,A -85,B 0,C 180,E1 18524.622,E2 18524.622} C_VEL
LIN {X 0,Y 543.549,Z 354.169,A -85,B 0,C 180,E1 18523.818,E2 18523.818} C_VEL
LIN {X 0,Y 545.348,Z 357.628,A -85,B 0,C 180,E1 18523.16,E2 18523.16} C_VEL
LIN {X 0,Y 548.225,Z 360.142,A -85,B 0,C 180,E1 18522.267,E2 18522.267} C_VEL
LIN {X 0,Y 549.404,Z 360.929,A -85,B 0,C 180,E1 18521.922,E2 18521.922} C_VEL
LIN {X 0,Y 551.761,Z 364.638,A -85,B 0,C 180,E1 18521.182,E2 18521.182} C_VEL
LIN {X 0,Y 555.012,Z 367.385,A -85,B 0,C 180,E1 18520.285,E2 18520.285} C_VEL
LIN {X 0,Y 558.035,Z 371.53,A -85,B 0,C 180,E1 18519.44,E2 18519.44} C_VEL
LIN {X 0,Y 560.363,Z 373.699,A -85,B 0,C 180,E1 18518.845,E2 18518.845} C_VEL
LIN {X 0,Y 563.794,Z 378.028,A -85,B 0,C 180,E1 18517.97,E2 18517.97} C_VEL
LIN {X 0,Y 565.638,Z 379.991,A -85,B 0,C 180,E1 18517.526,E2 18517.526} C_VEL
LIN {X 0,Y 569.473,Z 384.555,A -85,B 0,C 180,E1 18516.621,E2 18516.621} C_VEL
LIN {X 0,Y 576.123,Z 392.77,A -85,B 0,C 180,E1 18515.138,E2 18515.138} C_VEL
LIN {X 0,Y 580.705,Z 398.542,A -85,B 0,C 180,E1 18514.174,E2 18514.174} C_VEL
LIN {X 0,Y 586.519,Z 406.298,A -85,B 0,C 180,E1 18513.006,E2 18513.006} C_VEL
LIN {X 0,Y 596.123,Z 419.851,A -85,B 0,C 180,E1 18511.196,E2 18511.196} C_VEL
LIN {X 0,Y 605.205,Z 434.135,A -85,B 0,C 180,E1 18509.593,E2 18509.593} C_VEL
LIN {X 0,Y 596.828,Z 651.529,A -85,B 0,C 180,E1 18506.379,E2 18506.379} C_VEL
LIN {X 0,Y 590.769,Z 817.906,A -85,B 0,C 180,E1 18503.947,E2 18503.947} C_VEL
LIN {X 0,Y 589.101,Z 842.591,A -85,B 0,C 180,E1 18503.486,E2 18503.486} C_VEL
LIN {X 0,Y 586.482,Z 870.48,A -85,B 0,C 180,E1 18502.776,E2 18502.776} C_VEL
LIN {X 0,Y 584.576,Z 887.696,A -85,B 0,C 180,E1 18502.237,E2 18502.237} C_VEL
LIN {X 0,Y 582.934,Z 895.241,A -85,B 0,C 180,E1 18502.045,E2 18502.045} C_VEL
LIN {X 0,Y 576.254,Z 913.987,A -85,B 0,C 180,E1 18501.756,E2 18501.756} C_VEL
LIN {X 0,Y 574.586,Z 920.997,A -85,B 0,C 180,E1 18501.531,E2 18501.531} C_VEL
LIN {X 0,Y 570.522,Z 946.437,A -85,B 0,C 180,E1 18500.297,E2 18500.297} C_VEL
LIN {X 0,Y 567.03,Z 966.721,A -85,B 0,C 180,E1 18499.154,E2 18499.154} C_VEL
LIN {X 0,Y 563.554,Z 985.633,A -85,B 0,C 180,E1 18497.945,E2 18497.945} C_VEL
LIN {X 0,Y 559.811,Z 1004.939,A -85,B 0,C 180,E1 18496.555,E2 18496.555} C_VEL
LIN {X 0,Y 554.922,Z 1028.939,A -85,B 0,C 180,E1 18494.572,E2 18494.572} C_VEL
LIN {X 0,Y 551.036,Z 1047.452,A -85,B 0,C 180,E1 18492.814,E2 18492.814} C_VEL
LIN {X 0,Y 547.542,Z 1064.095,A -85,B 0,C 180,E1 18491.044,E2 18491.044} C_VEL
LIN {X 0,Y 544.104,Z 1080.698,A -85,B 0,C 180,E1 18489.073,E2 18489.073} C_VEL
LIN {X 0,Y 540.181,Z 1100.154,A -85,B 0,C 180,E1 18486.453,E2 18486.453} C_VEL
LIN {X 0,Y 537.467,Z 1114.171,A -85,B 0,C 180,E1 18484.309,E2 18484.309} C_VEL
LIN {X 0,Y 535.224,Z 1126.704,A -85,B 0,C 180,E1 18482.169,E2 18482.169} C_VEL
LIN {X 0,Y 533.093,Z 1139.7,A -85,B 0,C 180,E1 18479.68,E2 18479.68} C_VEL
LIN {X 0,Y 531.153,Z 1152.928,A -85,B 0,C 180,E1 18476.737,E2 18476.737} C_VEL
LIN {X 0,Y 529.979,Z 1162.296,A -85,B 0,C 180,E1 18474.32,E2 18474.32} C_VEL
LIN {X 0,Y 529.155,Z 1170.206,A -85,B 0,C 180,E1 18471.97,E2 18471.97} C_VEL
LIN {X 0,Y 528.572,Z 1177.474,A -85,B 0,C 180,E1 18469.446,E2 18469.446} C_VEL
LIN {X 0,Y 528.165,Z 1184.542,A -85,B 0,C 180,E1 18466.384,E2 18466.384} C_VEL
LIN {X 0,Y 527.995,Z 1189.026,A -85,B 0,C 180,E1 18463.804,E2 18463.804} C_VEL
LIN {X 0,Y 527.931,Z 1192.122,A -85,B 0,C 180,E1 18461.359,E2 18461.359} C_VEL
LIN {X 0,Y 527.913,Z 1194.075,A -85,B 0,C 180,E1 18458.934,E2 18458.934} C_VEL
LIN {X 0,Y 527.91,Z 1194.956,A -85,B 0,C 180,E1 18456.197,E2 18456.197} C_VEL
LIN {X 0,Y 527.91,Z 1194.252,A -85,B 0,C 180,E1 18453.257,E2 18453.257} C_VEL
LIN {X 0,Y 527.928,Z 1192.34,A -85,B 0,C 180,E1 18450.759,E2 18450.759} C_VEL
LIN {X 0,Y 527.979,Z 1189.414,A -85,B 0,C 180,E1 18448.372,E2 18448.372} C_VEL
LIN {X 0,Y 528.115,Z 1185.396,A -85,B 0,C 180,E1 18445.983,E2 18445.983} C_VEL
LIN {X 0,Y 528.456,Z 1179.268,A -85,B 0,C 180,E1 18443.154,E2 18443.154} C_VEL
LIN {X 0,Y 529.072,Z 1171.052,A -85,B 0,C 180,E1 18440.207,E2 18440.207} C_VEL
LIN {X 0,Y 529.904,Z 1163.048,A -85,B 0,C 180,E1 18437.799,E2 18437.799} C_VEL
LIN {X 0,Y 531,Z 1154.008,A -85,B 0,C 180,E1 18435.44,E2 18435.44} C_VEL
LIN {X 0,Y 532.611,Z 1142.702,A -85,B 0,C 180,E1 18432.857,E2 18432.857} C_VEL
LIN {X 0,Y 534.986,Z 1128.138,A -85,B 0,C 180,E1 18429.999,E2 18429.999} C_VEL
LIN {X 0,Y 537.231,Z 1115.402,A -85,B 0,C 180,E1 18427.801,E2 18427.801} C_VEL
LIN {X 0,Y 539.8,Z 1101.936,A -85,B 0,C 180,E1 18425.719,E2 18425.719} C_VEL
LIN {X 0,Y 543.169,Z 1085.369,A -85,B 0,C 180,E1 18423.428,E2 18423.428} C_VEL
LIN {X 0,Y 547.226,Z 1065.636,A -85,B 0,C 180,E1 18421.04,E2 18421.04} C_VEL
LIN {X 0,Y 550.69,Z 1049.075,A -85,B 0,C 180,E1 18419.262,E2 18419.262} C_VEL
LIN {X 0,Y 554.338,Z 1031.612,A -85,B 0,C 180,E1 18417.582,E2 18417.582} C_VEL
LIN {X 0,Y 558.928,Z 1009.497,A -85,B 0,C 180,E1 18415.701,E2 18415.701} C_VEL
LIN {X 0,Y 563.238,Z 987.266,A -85,B 0,C 180,E1 18414.076,E2 18414.076} C_VEL
LIN {X 0,Y 566.801,Z 967.913,A -85,B 0,C 180,E1 18412.829,E2 18412.829} C_VEL
LIN {X 0,Y 570.24,Z 947.957,A -85,B 0,C 180,E1 18411.695,E2 18411.695} C_VEL
LIN {X 0,Y 573.707,Z 926.279,A -85,B 0,C 180,E1 18410.625,E2 18410.625} C_VEL
LIN {X 0,Y 577.506,Z 899.37,A -85,B 0,C 180,E1 18409.514,E2 18409.514} C_VEL
LIN {X 0,Y 580.245,Z 876.361,A -85,B 0,C 180,E1 18408.738,E2 18408.738} C_VEL
LIN {X 0,Y 582.411,Z 855.045,A -85,B 0,C 180,E1 18408.148,E2 18408.148} C_VEL
LIN {X 0,Y 584.218,Z 833.3,A -85,B 0,C 180,E1 18407.668,E2 18407.668} C_VEL
LIN {X 0,Y 585.808,Z 806.164,A -85,B 0,C 180,E1 18407.211,E2 18407.211} C_VEL
LIN {X 0,Y 593.578,Z 580.141,A -85,B 0,C 180,E1 18403.951,E2 18403.951} C_VEL
LIN {X 0,Y 598.637,Z 437.808,A -85,B 0,C 180,E1 18401.857,E2 18401.857} C_VEL
LIN {X 0,Y 584.565,Z 417.617,A -85,B 0,C 180,E1 18399.612,E2 18399.612} C_VEL
LIN {X 0,Y 574.117,Z 403.151,A -85,B 0,C 180,E1 18397.81,E2 18397.81} C_VEL
LIN {X 0,Y 566.433,Z 393.358,A -85,B 0,C 180,E1 18396.41,E2 18396.41} C_VEL
LIN {X 0,Y 559.149,Z 384.138,A -85,B 0,C 180,E1 18395,E2 18395} C_VEL
LIN {X 0,Y 554.014,Z 377.979,A -85,B 0,C 180,E1 18393.958,E2 18393.958} C_VEL
LIN {X 0,Y 549.816,Z 372.799,A -85,B 0,C 180,E1 18393.064,E2 18393.064} C_VEL
LIN {X 0,Y 546.341,Z 368.807,A -85,B 0,C 180,E1 18392.304,E2 18392.304} C_VEL
LIN {X 0,Y 545.088,Z 367.077,A -85,B 0,C 180,E1 18392.015,E2 18392.015} C_VEL
LIN {X 0,Y 541.785,Z 363.792,A -85,B 0,C 180,E1 18391.269,E2 18391.269} C_VEL
LIN {X 0,Y 539.896,Z 360.926,A -85,B 0,C 180,E1 18390.803,E2 18390.803} C_VEL
LIN {X 0,Y 536.692,Z 358.092,A -85,B 0,C 180,E1 18390.046,E2 18390.046} C_VEL
LIN {X 0,Y 534.939,Z 354.807,A -85,B 0,C 180,E1 18389.568,E2 18389.568} C_VEL
LIN {X 0,Y 531.804,Z 352.735,A -85,B 0,C 180,E1 18388.803,E2 18388.803} C_VEL
LIN {X 0,Y 530.041,Z 349.876,A -85,B 0,C 180,E1 18388.306,E2 18388.306} C_VEL
LIN {X 0,Y 529.645,Z 348.216,A -85,B 0,C 180,E1 18388.142,E2 18388.142} C_VEL
LIN {X 0,Y 529.683,Z 348.209,A -85,B 0,C 180,E1 18384.772,E2 18384.772} C_VEL
LIN {X 0,Y 529.642,Z 348.196,A -85,B 0,C 180,E1 18381.484,E2 18381.484} C_VEL
LIN {X 0,Y 529.64,Z 348.234,A -85,B 0,C 180,E1 18378.036,E2 18378.036} C_VEL
LIN {X 0,Y 529.685,Z 348.182,A -85,B 0,C 180,E1 18374.764,E2 18374.764} C_VEL
LIN {X 0,Y 529.628,Z 348.23,A -85,B 0,C 180,E1 18371.434,E2 18371.434} C_VEL
LIN {X 0,Y 529.642,Z 348.242,A -85,B 0,C 180,E1 18368.031,E2 18368.031} C_VEL
LIN {X 0,Y 529.646,Z 348.237,A -85,B 0,C 180,E1 18364.873,E2 18364.873} C_VEL
LIN {X 0,Y 529.616,Z 348.241,A -85,B 0,C 180,E1 18361.515,E2 18361.515} C_VEL
LIN {X 0,Y 529.675,Z 348.235,A -85,B 0,C 180,E1 18358.269,E2 18358.269} C_VEL
LIN {X 0,Y 529.611,Z 348.244,A -85,B 0,C 180,E1 18355.018,E2 18355.018} C_VEL
LIN {X 0,Y 529.611,Z 348.243,A -85,B 0,C 180,E1 18351.532,E2 18351.532} C_VEL
LIN {X 0,Y 529.644,Z 348.222,A -85,B 0,C 180,E1 18348.346,E2 18348.346} C_VEL
LIN {X 0,Y 529.589,Z 348.206,A -85,B 0,C 180,E1 18345.121,E2 18345.121} C_VEL
LIN {X 0,Y 529.654,Z 348.213,A -85,B 0,C 180,E1 18341.965,E2 18341.965} C_VEL
LIN {X 0,Y 529.584,Z 348.218,A -85,B 0,C 180,E1 18338.746,E2 18338.746} C_VEL
LIN {X 0,Y 529.67,Z 348.317,A -85,B 0,C 180,E1 18337.934,E2 18337.934} C_VEL
LIN {X 0,Y 530.602,Z 351.196,A -85,B 0,C 180,E1 18337.625,E2 18337.625} C_VEL
LIN {X 0,Y 532.871,Z 353.77,A -85,B 0,C 180,E1 18337.027,E2 18337.027} C_VEL
LIN {X 0,Y 535.06,Z 355.101,A -85,B 0,C 180,E1 18336.5,E2 18336.5} C_VEL
LIN {X 0,Y 537.255,Z 358.774,A -85,B 0,C 180,E1 18335.918,E2 18335.918} C_VEL
LIN {X 0,Y 540.547,Z 361.806,A -85,B 0,C 180,E1 18335.142,E2 18335.142} C_VEL
LIN {X 0,Y 543.483,Z 365.734,A -85,B 0,C 180,E1 18334.442,E2 18334.442} C_VEL
LIN {X 0,Y 545.377,Z 367.864,A -85,B 0,C 180,E1 18334.012,E2 18334.012} C_VEL
LIN {X 0,Y 553.449,Z 377.971,A -85,B 0,C 180,E1 18332.247,E2 18332.247} C_VEL
LIN {X 0,Y 562.487,Z 389.78,A -85,B 0,C 180,E1 18330.413,E2 18330.413} C_VEL
LIN {X 0,Y 573.033,Z 404.129,A -85,B 0,C 180,E1 18328.434,E2 18328.434} C_VEL
LIN {X 0,Y 585.207,Z 421.375,A -85,B 0,C 180,E1 18326.327,E2 18326.327} C_VEL
LIN {X 0,Y 598.736,Z 441.262,A -85,B 0,C 180,E1 18324.169,E2 18324.169} C_VEL
LIN {X 0,Y 591.206,Z 652.816,A -85,B 0,C 180,E1 18321.082,E2 18321.082} C_VEL
LIN {X 0,Y 585.161,Z 825.878,A -85,B 0,C 180,E1 18318.576,E2 18318.576} C_VEL
LIN {X 0,Y 583.525,Z 849.933,A -85,B 0,C 180,E1 18318.137,E2 18318.137} C_VEL
LIN {X 0,Y 580.83,Z 878.732,A -85,B 0,C 180,E1 18317.418,E2 18317.418} C_VEL
LIN {X 0,Y 578.261,Z 900.854,A -85,B 0,C 180,E1 18316.716,E2 18316.716} C_VEL
LIN {X 0,Y 575.691,Z 920.419,A -85,B 0,C 180,E1 18315.976,E2 18315.976} C_VEL
LIN {X 0,Y 572.841,Z 939.822,A -85,B 0,C 180,E1 18315.126,E2 18315.126} C_VEL
LIN {X 0,Y 569.581,Z 960.013,A -85,B 0,C 180,E1 18314.111,E2 18314.111} C_VEL
LIN {X 0,Y 565.552,Z 983.36,A -85,B 0,C 180,E1 18312.758,E2 18312.758} C_VEL
LIN {X 0,Y 561.008,Z 1007.392,A -85,B 0,C 180,E1 18311.122,E2 18311.122} C_VEL
LIN {X 0,Y 557.317,Z 1026.059,A -85,B 0,C 180,E1 18309.675,E2 18309.675} C_VEL
LIN {X 0,Y 553.721,Z 1043.767,A -85,B 0,C 180,E1 18308.139,E2 18308.139} C_VEL
LIN {X 0,Y 549.96,Z 1062.204,A -85,B 0,C 180,E1 18306.348,E2 18306.348} C_VEL
LIN {X 0,Y 545.563,Z 1083.525,A -85,B 0,C 180,E1 18303.986,E2 18303.986} C_VEL
LIN {X 0,Y 542.427,Z 1098.814,A -85,B 0,C 180,E1 18302.065,E2 18302.065} C_VEL
LIN {X 0,Y 539.575,Z 1113.059,A -85,B 0,C 180,E1 18300.071,E2 18300.071} C_VEL
LIN {X 0,Y 537.051,Z 1126.464,A -85,B 0,C 180,E1 18297.981,E2 18297.981} C_VEL
LIN {X 0,Y 534.335,Z 1141.967,A -85,B 0,C 180,E1 18295.255,E2 18295.255} C_VEL
LIN {X 0,Y 532.295,Z 1154.738,A -85,B 0,C 180,E1 18292.649,E2 18292.649} C_VEL
LIN {X 0,Y 530.87,Z 1164.975,A -85,B 0,C 180,E1 18290.277,E2 18290.277} C_VEL
LIN {X 0,Y 529.754,Z 1174.318,A -85,B 0,C 180,E1 18287.805,E2 18287.805} C_VEL
LIN {X 0,Y 528.817,Z 1184.244,A -85,B 0,C 180,E1 18284.677,E2 18284.677} C_VEL
LIN {X 0,Y 528.341,Z 1190.818,A -85,B 0,C 180,E1 18282.127,E2 18282.127} C_VEL
LIN {X 0,Y 528.097,Z 1195.904,A -85,B 0,C 180,E1 18279.702,E2 18279.702} C_VEL
LIN {X 0,Y 527.973,Z 1200.002,A -85,B 0,C 180,E1 18277.181,E2 18277.181} C_VEL
LIN {X 0,Y 527.919,Z 1203.273,A -85,B 0,C 180,E1 18274.236,E2 18274.236} C_VEL
LIN {X 0,Y 527.909,Z 1204.69,A -85,B 0,C 180,E1 18271.52,E2 18271.52} C_VEL
LIN {X 0,Y 527.899,Z 1204.849,A -85,B 0,C 180,E1 18269.241,E2 18269.241} C_VEL
LIN {X 0,Y 527.916,Z 1203.97,A -85,B 0,C 180,E1 18266.852,E2 18266.852} C_VEL
LIN {X 0,Y 527.934,Z 1201.978,A -85,B 0,C 180,E1 18264.458,E2 18264.458} C_VEL
LIN {X 0,Y 528.005,Z 1198.724,A -85,B 0,C 180,E1 18261.945,E2 18261.945} C_VEL
LIN {X 0,Y 528.204,Z 1193.351,A -85,B 0,C 180,E1 18258.978,E2 18258.978} C_VEL
LIN {X 0,Y 528.632,Z 1186.67,A -85,B 0,C 180,E1 18256.213,E2 18256.213} C_VEL
LIN {X 0,Y 529.178,Z 1179.858,A -85,B 0,C 180,E1 18253.874,E2 18253.874} C_VEL
LIN {X 0,Y 530.029,Z 1171.891,A -85,B 0,C 180,E1 18251.523,E2 18251.523} C_VEL
LIN {X 0,Y 531.296,Z 1161.771,A -85,B 0,C 180,E1 18248.934,E2 18248.934} C_VEL
LIN {X 0,Y 533.288,Z 1148.285,A -85,B 0,C 180,E1 18245.993,E2 18245.993} C_VEL
LIN {X 0,Y 535.282,Z 1136.327,A -85,B 0,C 180,E1 18243.718,E2 18243.718} C_VEL
LIN {X 0,Y 537.551,Z 1123.668,A -85,B 0,C 180,E1 18241.565,E2 18241.565} C_VEL
LIN {X 0,Y 540.473,Z 1108.746,A -85,B 0,C 180,E1 18239.297,E2 18239.297} C_VEL
LIN {X 0,Y 544.208,Z 1090.047,A -85,B 0,C 180,E1 18236.804,E2 18236.804} C_VEL
LIN {X 0,Y 547.547,Z 1073.685,A -85,B 0,C 180,E1 18234.885,E2 18234.885} C_VEL
LIN {X 0,Y 550.891,Z 1057.435,A -85,B 0,C 180,E1 18233.172,E2 18233.172} C_VEL
LIN {X 0,Y 554.54,Z 1039.711,A -85,B 0,C 180,E1 18231.495,E2 18231.495} C_VEL
LIN {X 0,Y 559.305,Z 1016.203,A -85,B 0,C 180,E1 18229.539,E2 18229.539} C_VEL
LIN {X 0,Y 563.23,Z 995.698,A -85,B 0,C 180,E1 18228.06,E2 18228.06} C_VEL
LIN {X 0,Y 566.648,Z 976.98,A -85,B 0,C 180,E1 18226.862,E2 18226.862} C_VEL
LIN {X 0,Y 569.905,Z 957.948,A -85,B 0,C 180,E1 18225.782,E2 18225.782} C_VEL
LIN {X 0,Y 573.363,Z 936.421,A -85,B 0,C 180,E1 18224.714,E2 18224.714} C_VEL
LIN {X 0,Y 577.194,Z 910.048,A -85,B 0,C 180,E1 18223.606,E2 18223.606} C_VEL
LIN {X 0,Y 580.199,Z 885.521,A -85,B 0,C 180,E1 18222.771,E2 18222.771} C_VEL
LIN {X 0,Y 582.456,Z 864.142,A -85,B 0,C 180,E1 18222.175,E2 18222.175} C_VEL
LIN {X 0,Y 584.333,Z 842.667,A -85,B 0,C 180,E1 18221.696,E2 18221.696} C_VEL
LIN {X 0,Y 585.855,Z 818.566,A -85,B 0,C 180,E1 18221.28,E2 18221.28} C_VEL
LIN {X 0,Y 594.239,Z 596.558,A -85,B 0,C 180,E1 18218.02,E2 18218.02} C_VEL
LIN {X 0,Y 600.534,Z 441.398,A -85,B 0,C 180,E1 18215.703,E2 18215.703} C_VEL
LIN {X 0,Y 591.133,Z 426.517,A -85,B 0,C 180,E1 18213.989,E2 18213.989} C_VEL
LIN {X 0,Y 582.902,Z 414.583,A -85,B 0,C 180,E1 18212.386,E2 18212.386} C_VEL
LIN {X 0,Y 574.424,Z 402.947,A -85,B 0,C 180,E1 18210.607,E2 18210.607} C_VEL
LIN {X 0,Y 567.708,Z 394.094,A -85,B 0,C 180,E1 18209.086,E2 18209.086} C_VEL
LIN {X 0,Y 564.001,Z 389.321,A -85,B 0,C 180,E1 18208.195,E2 18208.195} C_VEL
LIN {X 0,Y 559.307,Z 383.368,A -85,B 0,C 180,E1 18207.006,E2 18207.006} C_VEL
LIN {X 0,Y 554.65,Z 377.572,A -85,B 0,C 180,E1 18205.751,E2 18205.751} C_VEL
LIN {X 0,Y 550.876,Z 373.135,A -85,B 0,C 180,E1 18204.675,E2 18204.675} C_VEL
LIN {X 0,Y 546.918,Z 368.137,A -85,B 0,C 180,E1 18203.459,E2 18203.459} C_VEL
LIN {X 0,Y 543.353,Z 364.927,A -85,B 0,C 180,E1 18202.334,E2 18202.334} C_VEL
LIN {X 0,Y 541.557,Z 361.666,A -85,B 0,C 180,E1 18201.67,E2 18201.67} C_VEL
LIN {X 0,Y 538.15,Z 359.438,A -85,B 0,C 180,E1 18200.502,E2 18200.502} C_VEL
LIN {X 0,Y 536.175,Z 356.271,A -85,B 0,C 180,E1 18199.699,E2 18199.699} C_VEL
LIN {X 0,Y 535.658,Z 355.039,A -85,B 0,C 180,E1 18199.463,E2 18199.463} C_VEL
LIN {X 0,Y 532.366,Z 353.308,A -85,B 0,C 180,E1 18198.167,E2 18198.167} C_VEL
LIN {X 0,Y 530.225,Z 350.503,A -85,B 0,C 180,E1 18197.165,E2 18197.165} C_VEL
LIN {X 0,Y 529.583,Z 348.205,A -85,B 0,C 180,E1 18196.734,E2 18196.734} C_VEL
LIN {X 0,Y 529.591,Z 348.24,A -85,B 0,C 180,E1 18193.206,E2 18193.206} C_VEL
LIN {X 0,Y 529.645,Z 348.215,A -85,B 0,C 180,E1 18189.892,E2 18189.892} C_VEL
LIN {X 0,Y 529.584,Z 348.211,A -85,B 0,C 180,E1 18186.722,E2 18186.722} C_VEL
LIN {X 0,Y 529.646,Z 348.25,A -85,B 0,C 180,E1 18183.463,E2 18183.463} C_VEL
LIN {X 0,Y 529.602,Z 348.2,A -85,B 0,C 180,E1 18180.216,E2 18180.216} C_VEL
LIN {X 0,Y 529.604,Z 348.24,A -85,B 0,C 180,E1 18176.753,E2 18176.753} C_VEL
LIN {X 0,Y 529.675,Z 348.211,A -85,B 0,C 180,E1 18173.388,E2 18173.388} C_VEL
LIN {X 0,Y 529.606,Z 348.207,A -85,B 0,C 180,E1 18170.107,E2 18170.107} C_VEL
LIN {X 0,Y 529.663,Z 348.373,A -85,B 0,C 180,E1 18168.981,E2 18168.981} C_VEL
LIN {X 0,Y 530.423,Z 350.863,A -85,B 0,C 180,E1 18168.529,E2 18168.529} C_VEL
LIN {X 0,Y 532.593,Z 353.492,A -85,B 0,C 180,E1 18167.532,E2 18167.532} C_VEL
LIN {X 0,Y 535.813,Z 355.361,A -85,B 0,C 180,E1 18166.263,E2 18166.263} C_VEL
LIN {X 0,Y 537.452,Z 358.508,A -85,B 0,C 180,E1 18165.564,E2 18165.564} C_VEL
LIN {X 0,Y 540.278,Z 361.056,A -85,B 0,C 180,E1 18164.544,E2 18164.544} C_VEL
LIN {X 0,Y 541.792,Z 362.014,A -85,B 0,C 180,E1 18164.039,E2 18164.039} C_VEL
LIN {X 0,Y 544.051,Z 365.71,A -85,B 0,C 180,E1 18163.229,E2 18163.229} C_VEL
LIN {X 0,Y 547.584,Z 368.688,A -85,B 0,C 180,E1 18162.135,E2 18162.135} C_VEL
LIN {X 0,Y 550.276,Z 372.521,A -85,B 0,C 180,E1 18161.294,E2 18161.294} C_VEL
LIN {X 0,Y 553.056,Z 374.961,A -85,B 0,C 180,E1 18160.515,E2 18160.515} C_VEL
LIN {X 0,Y 556.334,Z 379.232,A -85,B 0,C 180,E1 18159.594,E2 18159.594} C_VEL
LIN {X 0,Y 558.352,Z 381.263,A -85,B 0,C 180,E1 18159.068,E2 18159.068} C_VEL
LIN {X 0,Y 562.053,Z 385.73,A -85,B 0,C 180,E1 18158.118,E2 18158.118} C_VEL
LIN {X 0,Y 563.95,Z 388.088,A -85,B 0,C 180,E1 18157.647,E2 18157.647} C_VEL
LIN {X 0,Y 568.566,Z 393.584,A -85,B 0,C 180,E1 18156.554,E2 18156.554} C_VEL
LIN {X 0,Y 574.179,Z 400.564,A -85,B 0,C 180,E1 18155.295,E2 18155.295} C_VEL
LIN {X 0,Y 580.464,Z 408.543,A -85,B 0,C 180,E1 18153.971,E2 18153.971} C_VEL
LIN {X 0,Y 590.001,Z 422.039,A -85,B 0,C 180,E1 18152.084,E2 18152.084} C_VEL
LIN {X 0,Y 597.528,Z 433.457,A -85,B 0,C 180,E1 18150.695,E2 18150.695} C_VEL
LIN {X 0,Y 600.499,Z 438.483,A -85,B 0,C 180,E1 18150.16,E2 18150.16} C_VEL
LIN {X 0,Y 591.782,Z 654.732,A -85,B 0,C 180,E1 18146.944,E2 18146.944} C_VEL
LIN {X 0,Y 585.531,Z 818.081,A -85,B 0,C 180,E1 18144.539,E2 18144.539} C_VEL
LIN {X 0,Y 583.769,Z 843.081,A -85,B 0,C 180,E1 18144.068,E2 18144.068} C_VEL
LIN {X 0,Y 581.062,Z 870.639,A -85,B 0,C 180,E1 18143.361,E2 18143.361} C_VEL
LIN {X 0,Y 578.421,Z 892.791,A -85,B 0,C 180,E1 18142.644,E2 18142.644} C_VEL
LIN {X 0,Y 575.641,Z 913.356,A -85,B 0,C 180,E1 18141.851,E2 18141.851} C_VEL
LIN {X 0,Y 574.586,Z 920.997,A -85,B 0,C 180,E1 18141.531,E2 18141.531} C_VEL
LIN {X 0,Y 572.844,Z 928.162,A -85,B 0,C 180,E1 18141.286,E2 18141.286} C_VEL
LIN {X 0,Y 565.472,Z 946.33,A -85,B 0,C 180,E1 18140.819,E2 18140.819} C_VEL
LIN {X 0,Y 563.55,Z 953.219,A -85,B 0,C 180,E1 18140.521,E2 18140.521} C_VEL
LIN {X 0,Y 558.585,Z 979.947,A -85,B 0,C 180,E1 18138.902,E2 18138.902} C_VEL
LIN {X 0,Y 554.6,Z 999.791,A -85,B 0,C 180,E1 18137.508,E2 18137.508} C_VEL
LIN {X 0,Y 550.729,Z 1018.285,A -85,B 0,C 180,E1 18136.043,E2 18136.043} C_VEL
LIN {X 0,Y 546.648,Z 1037.357,A -85,B 0,C 180,E1 18134.341,E2 18134.341} C_VEL
LIN {X 0,Y 541.752,Z 1059.639,A -85,B 0,C 180,E1 18132.064,E2 18132.064} C_VEL
LIN {X 0,Y 538.017,Z 1076.532,A -85,B 0,C 180,E1 18130.091,E2 18130.091} C_VEL
LIN {X 0,Y 534.779,Z 1091.4,A -85,B 0,C 180,E1 18128.153,E2 18128.153} C_VEL
LIN {X 0,Y 531.464,Z 1107.513,A -85,B 0,C 180,E1 18125.81,E2 18125.81} C_VEL
LIN {X 0,Y 528.318,Z 1123.474,A -85,B 0,C 180,E1 18123.157,E2 18123.157} C_VEL
LIN {X 0,Y 526.116,Z 1135.598,A -85,B 0,C 180,E1 18120.872,E2 18120.872} C_VEL
LIN {X 0,Y 524.353,Z 1146.354,A -85,B 0,C 180,E1 18118.595,E2 18118.595} C_VEL
LIN {X 0,Y 522.848,Z 1156.793,A -85,B 0,C 180,E1 18116.093,E2 18116.093} C_VEL
LIN {X 0,Y 521.488,Z 1168.074,A -85,B 0,C 180,E1 18112.906,E2 18112.906} C_VEL
LIN {X 0,Y 520.786,Z 1175.338,A -85,B 0,C 180,E1 18110.452,E2 18110.452} C_VEL
LIN {X 0,Y 520.348,Z 1181.481,A -85,B 0,C 180,E1 18107.976,E2 18107.976} C_VEL
LIN {X 0,Y 520.085,Z 1186.681,A -85,B 0,C 180,E1 18105.385,E2 18105.385} C_VEL
LIN {X 0,Y 519.948,Z 1191.216,A -85,B 0,C 180,E1 18102.325,E2 18102.325} C_VEL
LIN {X 0,Y 519.915,Z 1193.672,A -85,B 0,C 180,E1 18099.631,E2 18099.631} C_VEL
LIN {X 0,Y 519.914,Z 1194.733,A -85,B 0,C 180,E1 18097.292,E2 18097.292} C_VEL
LIN {X 0,Y 519.903,Z 1194.804,A -85,B 0,C 180,E1 18094.964,E2 18094.964} C_VEL
LIN {X 0,Y 519.912,Z 1193.898,A -85,B 0,C 180,E1 18092.645,E2 18092.645} C_VEL
LIN {X 0,Y 519.943,Z 1191.867,A -85,B 0,C 180,E1 18090.22,E2 18090.22} C_VEL
LIN {X 0,Y 520.028,Z 1188.279,A -85,B 0,C 180,E1 18087.465,E2 18087.465} C_VEL
LIN {X 0,Y 520.287,Z 1182.478,A -85,B 0,C 180,E1 18084.375,E2 18084.375} C_VEL
LIN {X 0,Y 520.701,Z 1176.337,A -85,B 0,C 180,E1 18081.83,E2 18081.83} C_VEL
LIN {X 0,Y 521.361,Z 1169.274,A -85,B 0,C 180,E1 18079.39,E2 18079.39} C_VEL
LIN {X 0,Y 522.302,Z 1161.018,A -85,B 0,C 180,E1 18076.944,E2 18076.944} C_VEL
LIN {X 0,Y 523.942,Z 1149.125,A -85,B 0,C 180,E1 18073.935,E2 18073.935} C_VEL
LIN {X 0,Y 525.84,Z 1137.241,A -85,B 0,C 180,E1 18071.37,E2 18071.37} C_VEL
LIN {X 0,Y 527.886,Z 1125.607,A -85,B 0,C 180,E1 18069.139,E2 18069.139} C_VEL
LIN {X 0,Y 530.416,Z 1112.612,A -85,B 0,C 180,E1 18066.915,E2 18066.915} C_VEL
LIN {X 0,Y 534.185,Z 1094.223,A -85,B 0,C 180,E1 18064.143,E2 18064.143} C_VEL
LIN {X 0,Y 537.598,Z 1078.385,A -85,B 0,C 180,E1 18062.05,E2 18062.05} C_VEL
LIN {X 0,Y 541.055,Z 1062.688,A -85,B 0,C 180,E1 18060.19,E2 18060.19} C_VEL
LIN {X 0,Y 545.047,Z 1044.652,A -85,B 0,C 180,E1 18058.28,E2 18058.28} C_VEL
LIN {X 0,Y 550.068,Z 1021.515,A -85,B 0,C 180,E1 18056.142,E2 18056.142} C_VEL
LIN {X 0,Y 554.069,Z 1002.382,A -85,B 0,C 180,E1 18054.6,E2 18054.6} C_VEL
LIN {X 0,Y 557.773,Z 984.002,A -85,B 0,C 180,E1 18053.284,E2 18053.284} C_VEL
LIN {X 0,Y 561.314,Z 965.461,A -85,B 0,C 180,E1 18052.105,E2 18052.105} C_VEL
LIN {X 0,Y 564.989,Z 944.807,A -85,B 0,C 180,E1 18050.948,E2 18050.948} C_VEL
LIN {X 0,Y 569.269,Z 917.847,A -85,B 0,C 180,E1 18049.668,E2 18049.668} C_VEL
LIN {X 0,Y 572.335,Z 895.89,A -85,B 0,C 180,E1 18048.805,E2 18048.805} C_VEL
LIN {X 0,Y 574.898,Z 874.835,A -85,B 0,C 180,E1 18048.108,E2 18048.108} C_VEL
LIN {X 0,Y 577.092,Z 853.466,A -85,B 0,C 180,E1 18047.523,E2 18047.523} C_VEL
LIN {X 0,Y 579.127,Z 829.359,A -85,B 0,C 180,E1 18047.006,E2 18047.006} C_VEL
LIN {X 0,Y 580.895,Z 793.112,A -85,B 0,C 180,E1 18046.437,E2 18046.437} C_VEL
LIN {X 0,Y 588.946,Z 568.254,A -85,B 0,C 180,E1 18043.173,E2 18043.173} C_VEL
LIN {X 0,Y 593.596,Z 441.89,A -85,B 0,C 180,E1 18041.3,E2 18041.3} C_VEL
LIN {X 0,Y 577.281,Z 418.512,A -85,B 0,C 180,E1 18038.607,E2 18038.607} C_VEL
LIN {X 0,Y 568.288,Z 406.201,A -85,B 0,C 180,E1 18036.995,E2 18036.995} C_VEL
LIN {X 0,Y 559.019,Z 394.473,A -85,B 0,C 180,E1 18035.229,E2 18035.229} C_VEL
LIN {X 0,Y 555.338,Z 389.946,A -85,B 0,C 180,E1 18034.49,E2 18034.49} C_VEL
LIN {X 0,Y 551.377,Z 384.998,A -85,B 0,C 180,E1 18033.665,E2 18033.665} C_VEL
LIN {X 0,Y 546.913,Z 379.584,A -85,B 0,C 180,E1 18032.701,E2 18032.701} C_VEL
LIN {X 0,Y 543.302,Z 375.075,A -85,B 0,C 180,E1 18031.884,E2 18031.884} C_VEL
LIN {X 0,Y 538.909,Z 370.254,A -85,B 0,C 180,E1 18030.865,E2 18030.865} C_VEL
LIN {X 0,Y 537.527,Z 368.23,A -85,B 0,C 180,E1 18030.519,E2 18030.519} C_VEL
LIN {X 0,Y 534.188,Z 365.012,A -85,B 0,C 180,E1 18029.71,E2 18029.71} C_VEL
LIN {X 0,Y 532.404,Z 362.157,A -85,B 0,C 180,E1 18029.229,E2 18029.229} C_VEL
LIN {X 0,Y 529.165,Z 359.467,A -85,B 0,C 180,E1 18028.405,E2 18028.405} C_VEL
LIN {X 0,Y 527.205,Z 355.911,A -85,B 0,C 180,E1 18027.827,E2 18027.827} C_VEL
LIN {X 0,Y 523.763,Z 353.566,A -85,B 0,C 180,E1 18026.901,E2 18026.901} C_VEL
LIN {X 0,Y 522.058,Z 350.705,A -85,B 0,C 180,E1 18026.366,E2 18026.366} C_VEL
LIN {X 0,Y 521.706,Z 349.173,A -85,B 0,C 180,E1 18026.217,E2 18026.217} C_VEL
LIN {X 0,Y 521.752,Z 349.222,A -85,B 0,C 180,E1 18022.775,E2 18022.775} C_VEL
LIN {X 0,Y 521.706,Z 349.177,A -85,B 0,C 180,E1 18019.364,E2 18019.364} C_VEL
LIN {X 0,Y 521.695,Z 349.211,A -85,B 0,C 180,E1 18015.907,E2 18015.907} C_VEL
LIN {X 0,Y 521.74,Z 349.171,A -85,B 0,C 180,E1 18012.62,E2 18012.62} C_VEL
LIN {X 0,Y 521.692,Z 349.233,A -85,B 0,C 180,E1 18009.265,E2 18009.265} C_VEL
LIN {X 0,Y 521.691,Z 349.233,A -85,B 0,C 180,E1 18005.83,E2 18005.83} C_VEL
LIN {X 0,Y 521.734,Z 349.231,A -85,B 0,C 180,E1 18002.526,E2 18002.526} C_VEL
LIN {X 0,Y 521.677,Z 349.244,A -85,B 0,C 180,E1 17999.231,E2 17999.231} C_VEL
LIN {X 0,Y 521.695,Z 349.242,A -85,B 0,C 180,E1 17995.823,E2 17995.823} C_VEL
LIN {X 0,Y 521.694,Z 349.246,A -85,B 0,C 180,E1 17992.622,E2 17992.622} C_VEL
LIN {X 0,Y 521.665,Z 349.25,A -85,B 0,C 180,E1 17989.285,E2 17989.285} C_VEL
LIN {X 0,Y 521.711,Z 349.171,A -85,B 0,C 180,E1 17985.912,E2 17985.912} C_VEL
LIN {X 0,Y 521.661,Z 349.234,A -85,B 0,C 180,E1 17982.655,E2 17982.655} C_VEL
LIN {X 0,Y 521.716,Z 349.233,A -85,B 0,C 180,E1 17979.878,E2 17979.878} C_VEL
LIN {X 0,Y 522.568,Z 351.98,A -85,B 0,C 180,E1 17979.562,E2 17979.562} C_VEL
LIN {X 0,Y 524.844,Z 354.66,A -85,B 0,C 180,E1 17978.896,E2 17978.896} C_VEL
LIN {X 0,Y 527.273,Z 356.134,A -85,B 0,C 180,E1 17978.254,E2 17978.254} C_VEL
LIN {X 0,Y 529.218,Z 359.647,A -85,B 0,C 180,E1 17977.681,E2 17977.681} C_VEL
LIN {X 0,Y 532.352,Z 362.168,A -85,B 0,C 180,E1 17976.886,E2 17976.886} C_VEL
LIN {X 0,Y 535.786,Z 366.857,A -85,B 0,C 180,E1 17975.994,E2 17975.994} C_VEL
LIN {X 0,Y 538.139,Z 369.025,A -85,B 0,C 180,E1 17975.434,E2 17975.434} C_VEL
LIN {X 0,Y 541.26,Z 373.078,A -85,B 0,C 180,E1 17974.681,E2 17974.681} C_VEL
LIN {X 0,Y 547.35,Z 380.568,A -85,B 0,C 180,E1 17973.295,E2 17973.295} C_VEL
LIN {X 0,Y 551.888,Z 386.546,A -85,B 0,C 180,E1 17972.308,E2 17972.308} C_VEL
LIN {X 0,Y 559.08,Z 395.823,A -85,B 0,C 180,E1 17970.833,E2 17970.833} C_VEL
LIN {X 0,Y 570.093,Z 411.029,A -85,B 0,C 180,E1 17968.724,E2 17968.724} C_VEL
LIN {X 0,Y 581.791,Z 427.747,A -85,B 0,C 180,E1 17966.665,E2 17966.665} C_VEL
LIN {X 0,Y 593.706,Z 445.482,A -85,B 0,C 180,E1 17964.721,E2 17964.721} C_VEL
LIN {X 0,Y 585.755,Z 660.488,A -85,B 0,C 180,E1 17961.568,E2 17961.568} C_VEL
LIN {X 0,Y 579.756,Z 825.966,A -85,B 0,C 180,E1 17959.159,E2 17959.159} C_VEL
LIN {X 0,Y 578.037,Z 850.435,A -85,B 0,C 180,E1 17958.71,E2 17958.71} C_VEL
LIN {X 0,Y 575.26,Z 878.988,A -85,B 0,C 180,E1 17957.992,E2 17957.992} C_VEL
LIN {X 0,Y 572.597,Z 901.201,A -85,B 0,C 180,E1 17957.284,E2 17957.284} C_VEL
LIN {X 0,Y 569.865,Z 921.282,A -85,B 0,C 180,E1 17956.52,E2 17956.52} C_VEL
LIN {X 0,Y 566.902,Z 940.754,A -85,B 0,C 180,E1 17955.66,E2 17955.66} C_VEL
LIN {X 0,Y 563.193,Z 962.914,A -85,B 0,C 180,E1 17954.529,E2 17954.529} C_VEL
LIN {X 0,Y 558.376,Z 989.102,A -85,B 0,C 180,E1 17952.95,E2 17952.95} C_VEL
LIN {X 0,Y 554.468,Z 1008.76,A -85,B 0,C 180,E1 17951.577,E2 17951.577} C_VEL
LIN {X 0,Y 550.68,Z 1027.095,A -85,B 0,C 180,E1 17950.134,E2 17950.134} C_VEL
LIN {X 0,Y 546.903,Z 1044.886,A -85,B 0,C 180,E1 17948.568,E2 17948.568} C_VEL
LIN {X 0,Y 542.441,Z 1065.894,A -85,B 0,C 180,E1 17946.481,E2 17946.481} C_VEL
LIN {X 0,Y 538.332,Z 1084.659,A -85,B 0,C 180,E1 17944.335,E2 17944.335} C_VEL
LIN {X 0,Y 535.137,Z 1099.597,A -85,B 0,C 180,E1 17942.429,E2 17942.429} C_VEL
LIN {X 0,Y 532.258,Z 1113.361,A -85,B 0,C 180,E1 17940.479,E2 17940.479} C_VEL
LIN {X 0,Y 529.51,Z 1127.163,A -85,B 0,C 180,E1 17938.292,E2 17938.292} C_VEL
LIN {X 0,Y 526.448,Z 1143.686,A -85,B 0,C 180,E1 17935.299,E2 17935.299} C_VEL
LIN {X 0,Y 524.522,Z 1155.25,A -85,B 0,C 180,E1 17932.885,E2 17932.885} C_VEL
LIN {X 0,Y 523.032,Z 1165.394,A -85,B 0,C 180,E1 17930.488,E2 17930.488} C_VEL
LIN {X 0,Y 521.719,Z 1175.937,A -85,B 0,C 180,E1 17927.627,E2 17927.627} C_VEL
LIN {X 0,Y 520.832,Z 1184.847,A -85,B 0,C 180,E1 17924.68,E2 17924.68} C_VEL
LIN {X 0,Y 520.359,Z 1191.069,A -85,B 0,C 180,E1 17922.203,E2 17922.203} C_VEL
LIN {X 0,Y 520.103,Z 1196.108,A -85,B 0,C 180,E1 17919.74,E2 17919.74} C_VEL
LIN {X 0,Y 519.968,Z 1200.318,A -85,B 0,C 180,E1 17917.07,E2 17917.07} C_VEL
LIN {X 0,Y 519.917,Z 1203.422,A -85,B 0,C 180,E1 17914.081,E2 17914.081} C_VEL
LIN {X 0,Y 519.912,Z 1204.713,A -85,B 0,C 180,E1 17911.433,E2 17911.433} C_VEL
LIN {X 0,Y 519.905,Z 1204.826,A -85,B 0,C 180,E1 17909.119,E2 17909.119} C_VEL
LIN {X 0,Y 519.916,Z 1203.967,A -85,B 0,C 180,E1 17906.803,E2 17906.803} C_VEL
LIN {X 0,Y 519.936,Z 1201.975,A -85,B 0,C 180,E1 17904.372,E2 17904.372} C_VEL
LIN {X 0,Y 520.01,Z 1198.721,A -85,B 0,C 180,E1 17901.82,E2 17901.82} C_VEL
LIN {X 0,Y 520.227,Z 1193.351,A -85,B 0,C 180,E1 17898.807,E2 17898.807} C_VEL
LIN {X 0,Y 520.687,Z 1186.667,A -85,B 0,C 180,E1 17895.998,E2 17895.998} C_VEL
LIN {X 0,Y 521.311,Z 1179.599,A -85,B 0,C 180,E1 17893.54,E2 17893.54} C_VEL
LIN {X 0,Y 522.238,Z 1171.485,A -85,B 0,C 180,E1 17891.122,E2 17891.122} C_VEL
LIN {X 0,Y 523.775,Z 1160.382,A -85,B 0,C 180,E1 17888.264,E2 17888.264} C_VEL
